// TwinCAT 3 PLC project TcUnitVerifier
// Title: TcUnit verifier
// Company: www.tcunit.org
// Author: Jakob Sagatowski and contributors
// ProjectVersion: 1.2.1.0
// Description: This project is can be used to verify the different functions of TcUnit. It has various test suites to test different functions in TcUnit. By making sure to comment out everything except the test suite that is interesting it is possible to test only the specific function of TcUnit that is interesting.
// ProgramVersion: 3.1.4022.7
// libraries:
//   SysDir, * (System)
//   SysFile, * (System)
//   Tc2_Standard, * (Beckhoff Automation GmbH)
//   Tc2_System, * (Beckhoff Automation GmbH)
//   Tc3_Module, * (Beckhoff Automation GmbH)
//   TcUnit, * (www.tcunit.org)
//   Base Interfaces,newest,System
// project tree:
//   / PlcTask.TcTTO
//   POUs/ FB_ProtectedVariables.TcPOU
//   Test/ FB_AdjustAssertFailureMessageToMaxAllowedLengthTest.TcPOU, FB_TestDurationMeasurement.TcPOU, FB_AnyPrimitiveTypes.TcPOU, FB_AnyToUnionValue.TcPOU, FB_ArrayPrimitiveTypes.TcPOU, FB_AssertCountExceedsMaxNumber.TcPOU, FB_AssertEveryFailedTestTwice.TcPOU, FB_AssertEveryFailedTestTwiceArrayVersion.TcPOU, FB_AssertTrueFalse.TcPOU, FB_CheckIfSpecificTestIsFinished.TcPOU, FB_CreateDisabledTest.TcPOU, FB_CreateFourTestsWithSameName.TcPOU, FB_EmptyAssertionMessage.TcPOU, FB_EmptyTestSuite.TcPOU, FB_ExtendedTestInformation.TcPOU, FB_MultipleAssertWithSameParametersInDifferentCyclesAndInSameTest.TcPOU, FB_MultipleAssertWithSameParametersInDifferentCyclesButWithDifferentTests.TcPOU, FB_MultipleAssertWithSameParametersInSameCycleWithSameTest.TcPOU, FB_SkipAssertionsWhenFinished.TcPOU, FB_PrimitiveTypes.TcPOU, FB_TestFileControl.TcPOU, FB_TestFinishedNamed.TcPOU, FB_TestNumberOfAssertionsCalculation.TcPOU, FB_TestStreamBuffer.TcPOU, FB_TestXmlControl.TcPOU, FB_WriteProtectedFunctions.TcPOU, FB_TestFinishedNamedDoesNotExist.TcPOU, PRG_TEST.TcPOU
//   Version/ Global_Version.TcGVL
// real-time tasks:
//   TASK PlcTask: cycle T#10ms, priority 20, ADS port 350

CONFIGURATION TcUnitVerifier
    RESOURCE PLC ON TwinCAT3
        TASK PlcTask(INTERVAL := T#10ms, PRIORITY := 20);
        PROGRAM PRG_TEST WITH PlcTask : PRG_TEST;
    END_RESOURCE
END_CONFIGURATION

// ---- Version/Global_Version.TcGVL
{attribute 'TcGenerated'}
{attribute 'no-analysis'}
{attribute 'linkalways'}
// This function has been automatically generated from the project information.
VAR_GLOBAL CONSTANT
	{attribute 'const_non_replaced'}
	stLibVersion_TcUnit_verifier : ST_LibVersion := (iMajor := 1, iMinor := 2, iBuild := 1, iRevision := 0, nFlags := 0, sVersion := '1.2.1.0');
END_VAR

// ---- Test/PRG_TEST.TcPOU
PROGRAM PRG_TEST
VAR
    PrimitiveTypes : FB_PrimitiveTypes;
    (* The FB_ExtendedTestInformation needs to be instantiated as the second test suite in order to get ID=1 as
       test suite identity, which is verified by the .NET-verifier *)
    ExtendedTestInformation : FB_ExtendedTestInformation;
    AssertTrueFalse : FB_AssertTrueFalse;
    AssertEveryFailedTestTwice : FB_AssertEveryFailedTestTwice;
    CreateFourTestsWithSameName : FB_CreateFourTestsWithSameName;
    ArrayPrimitiveTypes : FB_ArrayPrimitiveTypes;
    CreateDisabledTest : FB_CreateDisabledTest;
    AnyPrimitiveTypes : FB_AnyPrimitiveTypes;
    AssertEveryFailedTestTwiceArrayVersion : FB_AssertEveryFailedTestTwiceArrayVersion;
    AnyToUnionValue : FB_AnyToUnionValue;
    MultipleAssertWithSameParametersInSameCycleWithSameTest : FB_MultipleAssertWithSameParametersInSameCycleWithSameTest;
    MultipleAssertWithSameParametersInDifferentCyclesButWithDifferentTests : FB_MultipleAssertWithSameParametersInDifferentCyclesButWithDifferentTests;
    MultipleAssertWithSameParametersInDifferentCyclesAndInSameTest : FB_MultipleAssertWithSameParametersInDifferentCyclesAndInSameTest;
    SkipAssertionsWhenFinished : FB_SkipAssertionsWhenFinished;
    AdjustAssertFailureMessageToMaxAllowedLengthTest : FB_AdjustAssertFailureMessageToMaxAllowedLengthTest;
    EmptyTestSuite : FB_EmptyTestSuite;
    CheckIfSpecificTestIsFinished : FB_CheckIfSpecificTestIsFinished;
    WriteProtectedFunctions : FB_WriteProtectedFunctions;
    TestNumberOfAssertionsCalculation : FB_TestNumberOfAssertionsCalculation;
    TestDurationMeasurement : FB_TestDurationMeasurement;
    TestFileControl : FB_TestFileControl;
    TestXmlControl : FB_TestXmlControl;
    TestStreamBuffer : FB_TestStreamBuffer;
    TestFinishedNamed : FB_TestFinishedNamed;
    EmptyAssertionMessage : FB_EmptyAssertionMessage;
    AssertCountExceedsMaxNumber : FB_AssertCountExceedsMaxNumber;
    (* The testsuite below is not active, as it will make TcUnit to abort. Uncomment if you want
       to test the function of where a test with a name that doesn't exist is set to finished *)
    //TestFinishedNamedDoesNotExist : FB_TestFinishedNamedDoesNotExist;
END_VAR

(* There are two ways to run TcUnit test suites:
    1. The RUN() will run all the test suites in parallel
    2. The RUN_IN_SEQUENCE() will run the test suites in sequence (one-by-one, next one doesn't start until the previous one is finished)
    Only use one of them at a time
*)

TcUnit.RUN();
//TcUnit.RUN_IN_SEQUENCE(T#0MS);

END_PROGRAM

// ---- Test/FB_PrimitiveTypes.TcPOU
(*
    This testsuite tests the different assert-functions for all the different data types in TwinCAT.
    For every data type at least two different tests have been defined:
        1. One test that succeeds (Expected and actual are equal)
        2. One test that fails (Expected and actual are false).
*)
FUNCTION_BLOCK FB_PrimitiveTypes EXTENDS TcUnit.FB_TestSuite

Test_ANY_Equals();
Test_ANY_Differ_DataType();
Test_BOOL_Equals();
Test_BOOL_Differ();
Test_BYTE_Equals();
Test_BYTE_Differ();
Test_DATE_AND_TIME_Equals();
Test_DATE_AND_TIME_Differ();
Test_DATE_Equals();
Test_DATE_Differ();
Test_DINT_Equals();
Test_DINT_Differ();
Test_DWORD_Equals();
Test_DWORD_Differ();
Test_INT_Equals();
Test_INT_Differ();
Test_LINT_Equals();
Test_LINT_Differ();
Test_LREAL_Equals();
Test_LREAL_Differ();
Test_LTIME_Equals();
Test_LTIME_Differ();
Test_LWORD_Equals();
Test_LWORD_Differ();
Test_REAL_Equals();
Test_REAL_Differ();
Test_SINT_Equals();
Test_SINT_Differ();
Test_STRING_Equals();
Test_STRING_Differ();
Test_STRING_Differ2();
Test_STRING_Differ3();
Test_TIME_Equals();
Test_TIME_Differ();
Test_TIME_OF_DAY_Equals();
Test_TIME_OF_DAY_Differ();
Test_UDINT_Equals();
Test_UDINT_Differ();
Test_UINT_Equals();
Test_UINT_Differ();
Test_ULINT_Equals();
Test_ULINT_Differ();
Test_USINT_Equals();
Test_USINT_Differ();
Test_WORD_Equals();
Test_WORD_Differ();
Test_WSTRING_Equals();
Test_WSTRING_Differ();

METHOD PRIVATE Test_ANY_Differ_DataType
VAR
    a : INT := 5;
    b : UINT := 5;
END_VAR
TEST('Test_ANY_Differ_DataType');

AssertEquals(Expected := a,
             Actual := b,
             Message := 'Values differ');

TEST_FINISHED();
END_METHOD

METHOD PRIVATE Test_ANY_Equals
VAR
    a : INT := 5;
    b : INT := 5;
END_VAR
TEST('Test_ANY_Equals');

AssertEquals(Expected := a,
             Actual := b,
             Message := 'Values differ');

TEST_FINISHED();
END_METHOD

METHOD PRIVATE Test_BOOL_Differ
VAR
    a : BOOL := TRUE;
    b : BOOL := FALSE;
END_VAR
TEST('Test_BOOL_Differ');

TCUNIT_ADSLOGSTR(msgCtrlMask := ADSLOG_MSGTYPE_ERROR,
                 msgFmtStr := 'This is just a string %s',
                 strArg := '2');

AssertEquals_BOOL(Expected := a,
                  Actual := b,
                  Message := 'Values differ');

TEST_FINISHED();
END_METHOD

METHOD PRIVATE Test_BOOL_Equals
VAR
    a : BOOL := TRUE;
    b : BOOL := TRUE;
END_VAR
TEST('Test_BOOL_Equals');

TCUNIT_ADSLOGSTR(msgCtrlMask := ADSLOG_MSGTYPE_ERROR,
                 msgFmtStr := 'This is just a string %s',
                 strArg := '1');

AssertEquals_BOOL(Expected := a,
                  Actual := b,
                  Message := 'Values differ');

TEST_FINISHED();
END_METHOD

METHOD PRIVATE Test_BYTE_Differ
VAR
    a : BYTE := 16#AB;
    b : BYTE := 16#CD;
END_VAR
TEST('Test_BYTE_Differ');

AssertEquals_BYTE(Expected := a,
                  Actual := b,
                  Message := 'Values differ');

TEST_FINISHED();
END_METHOD

METHOD PRIVATE Test_BYTE_Equals
VAR
    a : BYTE := 16#CD;
    b : BYTE := 16#CD;
END_VAR
TEST('Test_BYTE_Equals');

AssertEquals_BYTE(Expected := a,
                  Actual := b,
                  Message := 'Values differ');
TEST_FINISHED();
END_METHOD

METHOD PRIVATE Test_DATE_AND_TIME_Differ
VAR
    a : DATE_AND_TIME := DATE_AND_TIME#1996-05-06-15:36:30;
    b : DATE_AND_TIME := DATE_AND_TIME#1972-03-29-00:00:00;
END_VAR
TEST('Test_DATE_AND_TIME_Differ');

AssertEquals_DATE_AND_TIME(Expected := a,
                           Actual := b,
                           Message := 'Values differ');

TEST_FINISHED();
END_METHOD

METHOD PRIVATE Test_DATE_AND_TIME_Equals
VAR
    a : DATE_AND_TIME := DATE_AND_TIME#2019-01-20-13:54:30;
    b : DATE_AND_TIME := DATE_AND_TIME#2019-01-20-13:54:30;
END_VAR
TEST('Test_DATE_AND_TIME_Equals');

AssertEquals_DATE_AND_TIME(Expected := a,
                           Actual := b,
                           Message := 'Values differ');

TEST_FINISHED();
END_METHOD

METHOD PRIVATE Test_DATE_Differ
VAR
    a : DATE := DATE#1996-05-06;
    b : DATE := DATE#2019-01-20;
END_VAR
TEST('Test_DATE_Differ');

AssertEquals_DATE(Expected := a,
                  Actual := b,
                  Message := 'Values differ');

TEST_FINISHED();
END_METHOD

METHOD PRIVATE Test_DATE_Equals
VAR
    a : DATE := DATE#1996-05-06;
    b : DATE := DATE#1996-05-06;
END_VAR
TEST('Test_DATE_Equals');

AssertEquals_DATE(Expected := a,
                  Actual := b,
                  Message := 'Values differ');

TEST_FINISHED();
END_METHOD

METHOD PRIVATE Test_DINT_Differ
VAR
    a : DINT := -55555;
    b : DINT := 70000;
END_VAR
TEST('Test_DINT_Differ');

AssertEquals_DINT(Expected := a,
                  Actual := b,
                  Message := 'Values differ');

TEST_FINISHED();
END_METHOD

METHOD PRIVATE Test_DINT_Equals
VAR
    a : DINT := -80000;
    b : DINT := -80000;
END_VAR
TEST('Test_DINT_Equals');

AssertEquals_DINT(Expected := a,
                  Actual := b,
                  Message := 'Values differ');

TEST_FINISHED();
END_METHOD

METHOD PRIVATE Test_DWORD_Differ
VAR
    a : DWORD := 16#12345678;
    b : DWORD := 16#90ABCDEF;
END_VAR
TEST('Test_DWORD_Differ');

TCUNIT_ADSLOGSTR(msgCtrlMask := ADSLOG_MSGTYPE_HINT,
                 msgFmtStr := 'This is just a string %s',
                 strArg := '4');

AssertEquals_DWORD(Expected := a,
                   Actual := b,
                   Message := 'Values differ');

TEST_FINISHED();
END_METHOD

METHOD PRIVATE Test_DWORD_Equals
VAR
    a : DWORD := 16#7890ABCD;
    b : DWORD := 16#7890ABCD;
END_VAR
TEST('Test_DWORD_Equals');

TCUNIT_ADSLOGSTR(msgCtrlMask := ADSLOG_MSGTYPE_HINT,
                 msgFmtStr := 'This is just a string %s',
                 strArg := '3');

AssertEquals_DWORD(Expected := a,
                   Actual := b,
                   Message := 'Values differ');

TEST_FINISHED();
END_METHOD

METHOD PRIVATE Test_INT_Differ
VAR
    a : INT := -32000;
    b : INT := 15423;
END_VAR
TEST('Test_INT_Differ');

AssertEquals_INT(Expected := a,
                 Actual := b,
                 Message := 'Values differ');

TEST_FINISHED();
END_METHOD

METHOD PRIVATE Test_INT_Equals
VAR
    a : INT := -12345;
    b : INT := -12345;
END_VAR
TEST('Test_INT_Equals');

AssertEquals_INT(Expected := a,
                 Actual := b,
                 Message := 'Values differ');

TEST_FINISHED();
END_METHOD

METHOD PRIVATE Test_LINT_Differ
VAR
    a : LINT := -451416345;
    b : LINT := 589532453;
END_VAR
TEST('Test_LINT_Differ');

AssertEquals_LINT(Expected := a,
                  Actual := b,
                  Message := 'Values differ');

TEST_FINISHED();
END_METHOD

METHOD PRIVATE Test_LINT_Equals
VAR
    a : LINT := -123456789;
    b : LINT := -123456789;
END_VAR
TEST('Test_LINT_Equals');

AssertEquals_LINT(Expected := a,
                  Actual := b,
                  Message := 'Values differ');

TEST_FINISHED();
END_METHOD

METHOD PRIVATE Test_LREAL_Differ
VAR
    a : LREAL := 1234567.89;
    b : LREAL := 1234567.76;
    c : LREAL := 0.0;
END_VAR
TEST('Test_LREAL_Differ');

AssertEquals_LREAL(Expected := a,
                   Actual := b,
                   Delta := 0.1,
                   Message := 'Values a and b differ');

MEMSET (ADR(c), 255, SIZEOF(c));

AssertEquals_LREAL(Expected := a,
                   Actual := c,
                   Delta := 0.1,
                   Message := 'Values a and c differ');

TEST_FINISHED();
END_METHOD

METHOD PRIVATE Test_LREAL_Equals
VAR
    a : LREAL := 1234567.89;
    b : LREAL := 1234567.76;
END_VAR
TEST('Test_LREAL_Equals');

AssertEquals_LREAL(Expected := a,
                   Actual := b,
                   Delta := 0.2,
                   Message := 'Values differ');

TEST_FINISHED();
END_METHOD

METHOD PRIVATE Test_LTIME_Differ
VAR
    a : LTIME := LTIME#213503D23H34M33S709MS551US615NS;
    b : LTIME := LTIME#1000D15H23M12S34MS2US44NS;
END_VAR
TEST('Test_LTIME_Differ');

AssertEquals_LTIME(Expected := a,
                   Actual := b,
                   Message := 'Values differ');

TEST_FINISHED();
END_METHOD

METHOD PRIVATE Test_LTIME_Equals
VAR
    a : LTIME := LTIME#213503D23H34M33S709MS551US615NS;
    b : LTIME := LTIME#213503D23H34M33S709MS551US615NS;
END_VAR
TEST('Test_LTIME_Equals');

AssertEquals_LTIME(Expected := a,
                   Actual := b,
                   Message := 'Values differ');

TEST_FINISHED();
END_METHOD

METHOD PRIVATE Test_LWORD_Differ
VAR
    a : LWORD := 16#0123656789ABCBEC;
    b : LWORD := 16#0123256789ABCAEE;
END_VAR
TEST('Test_LWORD_Differ');

AssertEquals_LWORD(Expected := a,
                   Actual := b,
                   Message := 'Values differ');

TEST_FINISHED();
END_METHOD

METHOD PRIVATE Test_LWORD_Equals
VAR
    a : LWORD := 16#0123456789ABCDEF;
    b : LWORD := 16#0123456789ABCDEF;
END_VAR
TEST('Test_LWORD_Equals');

AssertEquals_LWORD(Expected := a,
                   Actual := b,
                   Message := 'Values differ');

TEST_FINISHED();
END_METHOD

METHOD PRIVATE Test_REAL_Differ
VAR
    a : REAL := 1234.5;
    b : REAL := 1234.4;
    c : REAL := 0.0;
END_VAR
TEST('Test_REAL_Differ');

TCUNIT_ADSLOGSTR(msgCtrlMask := ADSLOG_MSGTYPE_WARN,
                 msgFmtStr := 'This is just a string %s',
                 strArg := '6');

AssertEquals_REAL(Expected := a,
                  Actual := b,
                  Delta := 0.05,
                  Message := 'Values a and b differ');

MEMSET (ADR(c), 255, SIZEOF(c));

AssertEquals_REAL(Expected := a,
                  Actual := c,
                  Delta := 0.1,
                  Message := 'Values a and c differ');

TEST_FINISHED();
END_METHOD

METHOD PRIVATE Test_REAL_Equals
VAR
    a : REAL := 1234.5;
    b : REAL := 1234.4;
END_VAR
TEST('Test_REAL_Equals');

TCUNIT_ADSLOGSTR(msgCtrlMask := ADSLOG_MSGTYPE_WARN,
                 msgFmtStr := 'This is just a string %s',
                 strArg := '5');

AssertEquals_REAL(Expected := a,
                  Actual := b,
                  Delta := 0.1,
                  Message := 'Values differ');

TEST_FINISHED();
END_METHOD

METHOD PRIVATE Test_SINT_Differ
VAR
    a : SINT := 127;
    b : SINT := -30;
END_VAR
TEST('Test_SINT_Differ');

AssertEquals_SINT(Expected := a,
                  Actual := b,
                  Message := 'Values differ');

TEST_FINISHED();
END_METHOD

METHOD PRIVATE Test_SINT_Equals
VAR
    a : SINT := -128;
    b : SINT := -128;
END_VAR
TEST('Test_SINT_Equals');

AssertEquals_SINT(Expected := a,
                  Actual := b,
                  Message := 'Values differ');

TEST_FINISHED();
END_METHOD

METHOD PRIVATE Test_STRING_Differ
VAR
    a : STRING := 'This is a string';
    b : STRING := 'This is another string';
END_VAR
TEST('Test_STRING_Differ');

AssertEquals_STRING(Expected := a,
                    Actual := b,
                    Message := 'Values differ');

TEST_FINISHED();
END_METHOD

METHOD PRIVATE Test_STRING_Differ2
VAR
    a : STRING := '';
    b : STRING := 'This string is not empty';
END_VAR
TEST('Test_STRING_Differ2');

AssertEquals_STRING(Expected := a,
                    Actual := b,
                    Message := 'Values differ');

TEST_FINISHED();
END_METHOD

METHOD PRIVATE Test_STRING_Differ3
VAR
    a : STRING := 'This string is not empty';
    b : STRING := '';
END_VAR
TEST('Test_STRING_Differ3');

AssertEquals_STRING(Expected := a,
                    Actual := b,
                    Message := 'Values differ');

TEST_FINISHED();
END_METHOD

METHOD PRIVATE Test_STRING_Equals
VAR
    a : STRING := 'Hello there';
    b : STRING := 'Hello there';
END_VAR
TEST('Test_STRING_Equals');

AssertEquals_STRING(Expected := a,
                    Actual := b,
                    Message := 'Values differ');

TEST_FINISHED();
END_METHOD

METHOD PRIVATE Test_TIME_Differ
VAR
    a : TIME := T#12H34M15S10MS;
    b : TIME := T#11H34M13S244MS;
END_VAR
TEST('Test_TIME_Differ');

AssertEquals_TIME(Expected := a,
                  Actual := b,
                  Message := 'Values differ');

TEST_FINISHED();
END_METHOD

METHOD PRIVATE Test_TIME_Equals
VAR
    a : TIME := T#11H34M13S244MS;
    b : TIME := T#11H34M13S244MS;
END_VAR
TEST('Test_TIME_Equals');

AssertEquals_TIME(Expected := a,
                  Actual := b,
                  Message := 'Values differ');

TEST_FINISHED();
END_METHOD

METHOD PRIVATE Test_TIME_OF_DAY_Differ
VAR
    a : TIME_OF_DAY := TIME_OF_DAY#15:36:30.123;
    b : TIME_OF_DAY := TIME_OF_DAY#06:21:11.492;
END_VAR
TEST('Test_TIME_OF_DAY_Differ');

AssertEquals_TIME_OF_DAY(Expected := a,
                         Actual := b,
                         Message := 'Values differ');

TEST_FINISHED();
END_METHOD

METHOD PRIVATE Test_TIME_OF_DAY_Equals
VAR
    a : TIME_OF_DAY := TIME_OF_DAY#06:21:11.492;
    b : TIME_OF_DAY := TIME_OF_DAY#06:21:11.492;
END_VAR
TEST('Test_TIME_OF_DAY_Equals');

AssertEquals_TIME_OF_DAY(Expected := a,
                         Actual := b,
                         Message := 'Values differ');

TEST_FINISHED();
END_METHOD

METHOD PRIVATE Test_UDINT_Differ
VAR
    a : UDINT := 34124214;
    b : UDINT := 52343244;
END_VAR
TEST('Test_UDINT_Differ');

AssertEquals_UDINT(Expected := a,
                   Actual := b,
                   Message := 'Values differ');

TEST_FINISHED();
END_METHOD

METHOD PRIVATE Test_UDINT_Equals
VAR
    a : UDINT := 21845123;
    b : UDINT := 21845123;
END_VAR
TEST('Test_UDINT_Equals');

AssertEquals_UDINT(Expected := a,
                   Actual := b,
                   Message := 'Values differ');

TEST_FINISHED();
END_METHOD

METHOD PRIVATE Test_UINT_Differ
VAR
    a : UINT := 64322;
    b : UINT := 32312;
END_VAR
TEST('Test_UINT_Differ');

AssertEquals_UINT(Expected := a,
                  Actual := b,
                  Message := 'Values differ');

TEST_FINISHED();
END_METHOD

METHOD PRIVATE Test_UINT_Equals
VAR
    a : UINT := 65535;
    b : UINT := 65535;
END_VAR
TEST('Test_UINT_Equals');

AssertEquals_UINT(Expected := a,
                  Actual := b,
                  Message := 'Values differ');

TEST_FINISHED();
END_METHOD

METHOD PRIVATE Test_ULINT_Differ
VAR
    a : ULINT := 10000;
    b : ULINT := 53685437234;
END_VAR
TEST('Test_ULINT_Differ');

AssertEquals_ULINT(Expected := a,
                   Actual := b,
                   Message := 'Values differ');

TEST_FINISHED();
END_METHOD

METHOD PRIVATE Test_ULINT_Equals
VAR
    a : ULINT := 45683838383;
    b : ULINT := 45683838383;
END_VAR
TEST('Test_ULINT_Equals');

AssertEquals_ULINT(Expected := a,
                   Actual := b,
                   Message := 'Values differ');

TEST_FINISHED();
END_METHOD

METHOD PRIVATE Test_USINT_Differ
VAR
    a : USINT := 3;
    b : USINT := 7;
END_VAR
TEST('Test_USINT_Differ');

AssertEquals_USINT(Expected := a,
                   Actual := b,
                   Message := 'Values differ');

TEST_FINISHED();
END_METHOD

METHOD PRIVATE Test_USINT_Equals
VAR
    a : USINT := 5;
    b : USINT := 5;
END_VAR
TEST('Test_USINT_Equals');

AssertEquals_USINT(Expected := a,
                   Actual := b,
                   Message := 'Values differ');

TEST_FINISHED();
END_METHOD

METHOD PRIVATE Test_WORD_Differ
VAR
    a : WORD := 16#EF01;
    b : WORD := 16#2345;
END_VAR
TEST('Test_WORD_Differ');

AssertEquals_WORD(Expected := a,
                  Actual := b,
                  Message := 'Values differ');

TEST_FINISHED();
END_METHOD

METHOD PRIVATE Test_WORD_Equals
VAR
    a : WORD := 16#ABCD;
    b : WORD := 16#ABCD;
END_VAR
TEST('Test_WORD_Equals');

AssertEquals_WORD(Expected := a,
                  Actual := b,
                  Message := 'Values differ');

TEST_FINISHED();
END_METHOD

METHOD PRIVATE Test_WSTRING_Differ
VAR
    a : WSTRING := "äö";
    b : WSTRING := "æåŅ";
END_VAR
TEST('Test_WSTRING_Differ');

AssertEquals_WSTRING(Expected := a,
                     Actual := b,
                     Message := 'Values differ');

TEST_FINISHED();
END_METHOD

METHOD PRIVATE Test_WSTRING_Equals
VAR
    a : WSTRING := "ŏŜŢ";
    b : WSTRING := "ŏŜŢ";
END_VAR
TEST('Test_WSTRING_Equals');

AssertEquals_WSTRING(Expected := a,
                     Actual := b,
                     Message := 'Values differ');

TEST_FINISHED();
END_METHOD

END_FUNCTION_BLOCK

// ---- Test/FB_ExtendedTestInformation.TcPOU
(* This test suite makes sure to create different variants of tests that will produce various extended logs, i.e. the
   ADS-logs that provide information on how many tests have finished/are successful within the test suites.
   This test suite needs to be instantiated as the second test suite in the order in order to get the ID=1 as identity. *)
FUNCTION_BLOCK FB_ExtendedTestInformation EXTENDS TcUnit.FB_TestSuite

Test_ExtendedTestInformation_BOOL_AssertFailed();
Test_ExtendedTestInformation_BOOL_AssertSuccess();
Test_ExtendedTestInformation_BYTE_TwoFailedAsserts();
Test_ExtendedTestInformation_LINT_AssertFailed();
Test_ExtendedTestInformation_LINT_AssertSuccess();

METHOD PRIVATE Test_ExtendedTestInformation_BOOL_AssertFailed
VAR
    a : BOOL := TRUE;
    b : BOOL := FALSE;
END_VAR
TEST('Test_ExtendedTestInformation_BOOL_AssertFailed');

AssertEquals_BOOL(Expected := a,
                  Actual := b,
                  Message := 'Extendedinformation values differ BOOL failure');

TEST_FINISHED();
END_METHOD

METHOD PRIVATE Test_ExtendedTestInformation_BOOL_AssertSuccess
VAR
    a : BOOL := TRUE;
    b : BOOL := TRUE;
END_VAR
TEST('Test_ExtendedTestInformation_BOOL_AssertSuccess');

AssertEquals_BOOL(Expected := a,
                  Actual := b,
                  Message := 'Extendedinformation values differ BOOL success');

TEST_FINISHED();
END_METHOD

METHOD PRIVATE Test_ExtendedTestInformation_BYTE_TwoFailedAsserts
VAR
    a : BYTE := 16#AB;
    b : BYTE := 16#CD;
    c : BYTE := 16#EF;
    d : BYTE := 16#01;
END_VAR
TEST('Test_ExtendedTestInformation_BYTE_TwoFailedAsserts');

AssertEquals_BYTE(Expected := a,
                  Actual := b,
                  Message := 'Extendedinformation values differ BYTE1');

AssertEquals_BYTE(Expected := c,
                  Actual := d,
                  Message := 'Extendedinformation values differ BYTE2');

TEST_FINISHED();
END_METHOD

METHOD PRIVATE Test_ExtendedTestInformation_LINT_AssertFailed
VAR
    a : LINT := -451416345;
    b : LINT := 589532453;
END_VAR
TEST('Test_ExtendedTestInformation_LINT_AssertFailed');

AssertEquals_LINT(Expected := a,
                  Actual := b,
                  Message := 'Extendedinformation values differ LINT failure');

TEST_FINISHED();
END_METHOD

METHOD PRIVATE Test_ExtendedTestInformation_LINT_AssertSuccess
VAR
    a : LINT := -123456789;
    b : LINT := -123456789;
END_VAR
TEST('Test_ExtendedTestInformation_LINT_AssertSuccess');

AssertEquals_LINT(Expected := a,
                  Actual := b,
                  Message := 'Extendedinformation values differ LINT success');

TEST_FINISHED();
END_METHOD

END_FUNCTION_BLOCK

// ---- Test/FB_AssertTrueFalse.TcPOU
(* 
    This testsuite verifies that the Assert_True and Assert_False methods do what they are supposed to. It does so
    by making sure that every assert-method (assert_true & assert_false) does both one failing and one successful
    assert.
*)
FUNCTION_BLOCK FB_AssertTrueFalse EXTENDS TcUnit.FB_TestSuite

AssertThatINTsAreEqual();
AssertThatINTsAreNotEqual();
AssertThatWORDsAreEqual();
AssertThatWORDsAreNotEqual();

METHOD PRIVATE AssertThatINTsAreEqual
VAR
    a : INT := -33;
    b : INT := -44;
END_VAR
TEST('AssertThatINTsAreEqual');

AssertFalse(Condition := (a <> b),
            Message := 'INTs are equal');

TEST_FINISHED();
END_METHOD

METHOD PRIVATE AssertThatINTsAreNotEqual
VAR
    a : INT := -33;
    b : INT := -44;
END_VAR
TEST('AssertThatINTsAreNotEqual');

AssertFalse(Condition := (a = b),
            Message := 'INTs are equal');

TEST_FINISHED();
END_METHOD

METHOD PRIVATE AssertThatWORDsAreEqual
VAR
    a : WORD := 16#ABCD;
    b : WORD := 16#0123;
END_VAR
TEST('AssertThatWORDsAreEqual');

AssertTrue(Condition := (a = b),
           Message := 'WORDs are not equal');

TEST_FINISHED();
END_METHOD

METHOD PRIVATE AssertThatWORDsAreNotEqual
VAR
    a : WORD := 16#ABCD;
    b : WORD := 16#0123;
END_VAR
TEST('AssertThatWORDsAreNotEqual');

AssertTrue(Condition := (a <> b),
           Message := 'WORDs are equal');

TEST_FINISHED();
END_METHOD

END_FUNCTION_BLOCK

// ---- Test/FB_AssertEveryFailedTestTwice.TcPOU
(*
    In this testsuite we are running the same testcase over two cycles, and thus calling every assert method twice.
    This is in order to verify that we don't print every FAILED assert twice.
*)
FUNCTION_BLOCK FB_AssertEveryFailedTestTwice EXTENDS TcUnit.FB_TestSuite
VAR
    AssertCount : USINT := 0;
END_VAR

TwiceAssertCall();

METHOD PRIVATE TwiceAssertCall
VAR
    aANY : INT := 55;
    bANY : INT := 77;

    aBOOL : BOOL := TRUE;
    bBOOL : BOOL := FALSE;

    aBYTE : BYTE := 16#AB;
    bBYTE : BYTE := 16#BA;

    aDATE : DATE := DATE#1996-05-06;
    bDATE : DATE := DATE#2019-01-20;

    aDATE_AND_TIME : DATE_AND_TIME := DATE_AND_TIME#1996-05-06-15:36:30;
    bDATE_AND_TIME : DATE_AND_TIME := DATE_AND_TIME#1972-03-29-00:00:00;

    aDINT : DINT := 4444;
    bDINT : DINT := 3333;

    aDWORD : DWORD := 16#AAAAAAAA;
    bDWORD : DWORD := 16#BBBBBBBB;

    aINT : INT := 30000;
    bINT : INT := 32000;

    aLINT : LINT := 50000;
    bLINT : LINT := 50001;

    aLREAL : LREAL := 33.3;
    bLREAL : LREAL := 44.4;

    aLTIME : LTIME := LTIME#213503D23H34M33S709MS551US615NS;
    bLTIME : LTIME := LTIME#1000D15H23M12S34MS2US44NS;

    aLWORD : LWORD := 16#AAAAAAAAAAAAAAAA;
    bLWORD : LWORD := 16#BBBBBBBBBBBBBBBB;

    aREAL : REAL := 44.4;
    bREAL : REAL := 22.2;

    aSINT : SINT := 99;
    bSINT : SINT := 10;

    aSTRING : STRING := 'Hello world';
    bSTRING : STRING := 'Hey there';

    aUDINT : UDINT := 249494994;
    bUDINT : UDINT := 1223;

    aUINT : UINT := 3444;
    bUINT : UINT := 3445;

    aULINT : ULINT := 789234475;
    bULINT : ULINT := 34523327234;

    aUSINT : USINT := 34;
    bUSINT : USINT := 36;

    aTIME : TIME := T#12H34M15S10MS;
    bTIME : TIME := T#11H34M13S244MS;

    aTIME_OF_DAY : TIME_OF_DAY := TIME_OF_DAY#15:36:30.123;
    bTIME_OF_DAY : TIME_OF_DAY := TIME_OF_DAY#06:21:11.492;

    aWORD : WORD := 16#ABCD;
    bWORD : WORD := 16#89EF;

	aWSTRING : WSTRING := "åäöĦ";
    bWSTRING : WSTRING := "åäöŅ";
END_VAR
TEST('TwiceAssertCall');

AssertEquals(Expected := aANY,
             Actual := bANY,
             Message := 'Not equal ANY');

AssertEquals_BOOL(Expected := aBOOL,
                  Actual := bBOOL,
                  Message := 'Not equal BOOL');

AssertEquals_BYTE(Expected := aBYTE,
                  Actual := bBYTE,
                  Message := 'Not equal BYTE');

AssertEquals_DATE(Expected := aDATE,
                  Actual := bDATE,
                  Message := 'Not equal DATE');

AssertEquals_DATE_AND_TIME(Expected := aDATE_AND_TIME,
                           Actual := bDATE_AND_TIME,
                           Message := 'Not equal DATE_AND_TIME');

AssertEquals_DINT(Expected := aDINT,
                  Actual := bDINT,
                  Message := 'Not equal DINT');

AssertEquals_DWORD(Expected := aDWORD,
                   Actual := bDWORD,
                   Message := 'Not equal DWORD');

AssertEquals_INT(Expected := aINT,
                 Actual := bINT,
                 Message := 'Not equal INT');

AssertEquals_LINT(Expected := aLINT,
                  Actual := bLINT,
                  Message := 'Not equal LINT');

AssertEquals_LREAL(Expected := aLREAL,
                   Actual := bLREAL,
                   Delta := 0.1,
                   Message := 'Not equal LREAL');

AssertEquals_LTIME(Expected := aLTIME,
                   Actual := bLTIME,
                   Message := 'Not equal LTIME');

AssertEquals_LWORD(Expected := aLWORD,
                   Actual := bLWORD,
                   Message := 'Not equal LWORD');

AssertEquals_REAL(Expected := aREAL,
                  Actual := bREAL,
                  Delta := 0.1,
                  Message := 'Not equal REAL');

AssertEquals_SINT(Expected := aSINT,
                  Actual := bSINT,
                  Message := 'Not equal SINT');

AssertEquals_STRING(Expected := aSTRING,
                    Actual := bSTRING,
                    Message := 'Not equal STRING');

AssertEquals_UDINT(Expected := aUDINT,
                   Actual := bUDINT,
                   Message := 'Not equal UDINT');

AssertEquals_UINT(Expected := aUINT,
                  Actual := bUINT,
                  Message := 'Not equal UINT');

AssertEquals_ULINT(Expected := aULINT,
                   Actual := bULINT,
                   Message := 'Not equal ULINT');

AssertEquals_USINT(Expected := aUSINT,
                   Actual := bUSINT,
                   Message := 'Not equal USINT');

AssertEquals_TIME(Expected := aTIME,
                  Actual := bTIME,
                  Message := 'Not equal TIME');

AssertEquals_TIME_OF_DAY(Expected := aTIME_OF_DAY,
                         Actual := bTIME_OF_DAY,
                         Message := 'Not equal TIME_OF_DAY');

AssertEquals_WORD(Expected := aWORD,
                  Actual := bWORD,
                  Message := 'Not equal WORD');

AssertEquals_WSTRING(Expected := aWSTRING,
                     Actual := bWSTRING,
                     Message := 'Not equal WSTRING');

AssertCount := AssertCount + 1;
IF AssertCount = 2 THEN
    TEST_FINISHED();
END_IF
END_METHOD

END_FUNCTION_BLOCK

// ---- Test/FB_CreateFourTestsWithSameName.TcPOU
(*
    This testsuite creates four tests in the same testsuite with the same name. Every test in a testsuite should have
    an unique name. Every assert should be ignored if a duplicate test is being run.
*)
FUNCTION_BLOCK FB_CreateFourTestsWithSameName EXTENDS TcUnit.FB_TestSuite

TestOne();
TestOne_Again();
TestOne_AgainAgain();
TestOne_AgainAgainAgain();

METHOD PRIVATE TestOne
VAR
    a : INT := 55;
    b : INT := 55;
END_VAR
TEST('TestOne');

AssertEquals_INT(Expected := a,
                 Actual := b,
                 Message := 'A does not equal B');

TEST_FINISHED();
END_METHOD

METHOD PRIVATE TestOne_Again
VAR
    a : INT := 55;
    b : INT := 54;
END_VAR
TEST('TestOne');

AssertEquals_INT(Expected := a,
                 Actual := b,
                 Message := 'A does not equal B again');

TEST_FINISHED();
END_METHOD

METHOD PRIVATE TestOne_AgainAgain
VAR
    a : INT := 55;
    b : INT := 55;
END_VAR
TEST('TestOne');

AssertEquals_INT(Expected := a,
                 Actual := b,
                 Message := 'A does not equal B again');

TEST_FINISHED();
END_METHOD

METHOD PRIVATE TestOne_AgainAgainAgain
VAR
    a : INT := 55;
    b : INT := 55;
END_VAR
TEST('TestOne');

AssertEquals_INT(Expected := a,
                 Actual := b,
                 Message := 'A does not equal B again');

TEST_FINISHED();
END_METHOD

END_FUNCTION_BLOCK

// ---- Test/FB_ArrayPrimitiveTypes.TcPOU
(*
    This testsuite tests the different assert-functions for all the different type of arrays (varying by the different
    data types that are available in TwinCAT). For every type of array (BOOL, BYTE, INT etc.) at least three different
    tests have been defined:
        1. One test that succeeds, where the data and size of the arrays are matching
        2. One test that fails, where the size of the arrays differs
        3. One test that fails, where the content of the array differs
*)
FUNCTION_BLOCK FB_ArrayPrimitiveTypes EXTENDS TcUnit.FB_TestSuite

Test_BOOL_Array_Equals();
Test_BOOL_Array_DifferInSize();
Test_BOOL_Array_DifferInContent();
Test_BYTE_Array_Equals();
Test_BYTE_Array_DifferInSize();
Test_BYTE_Array_DifferInContent();
Test_DINT_Array_Equals();
Test_DINT_Array_DifferInSize();
Test_DINT_Array_DifferInContent();
Test_DWORD_Array_Equals();
Test_DWORD_Array_DifferInSize();
Test_DWORD_Array_DifferInContent();
Test_INT_Array_Equals();
Test_INT_Array_DifferInSize();
Test_INT_Array_DifferInContent();
Test_LINT_Array_Equals();
Test_LINT_Array_DifferInSize();
Test_LINT_Array_DifferInContent();
Test_LREAL_Array_Equals();
Test_LREAL_Array_DifferInSize();
Test_LREAL_Array_DifferInContent();
Test_LREAL_Array2d_Equals();
Test_LREAL_Array2d_DifferInSize_D1();
Test_LREAL_Array2d_DifferInSize_D2();
Test_LREAL_Array2d_DifferInContent_LBOUND();
Test_LREAL_Array2d_DifferInContent_Middle();
Test_LREAL_Array2d_DifferInContent_UBOUND();
Test_LREAL_Array3d_Equals();
Test_LREAL_Array3d_DifferInSize_D1();
Test_LREAL_Array3d_DifferInSize_D2();
Test_LREAL_Array3d_DifferInSize_D3();
Test_LREAL_Array3d_DifferInContent_LBOUND();
Test_LREAL_Array3d_DifferInContent_Middle();
Test_LREAL_Array3d_DifferInContent_UBOUND();
Test_LWORD_Array_Equals();
Test_LWORD_Array_DifferInSize();
Test_LWORD_Array_DifferInContent();
Test_REAL_Array_Equals();
Test_REAL_Array_DifferInSize();
Test_REAL_Array_DifferInContent();
Test_REAL_Array2d_Equals();
Test_REAL_Array2d_DifferInSize_D1();
Test_REAL_Array2d_DifferInSize_D2();
Test_REAL_Array2d_DifferInContent_LBOUND();
Test_REAL_Array2d_DifferInContent_Middle();
Test_REAL_Array2d_DifferInContent_UBOUND();
Test_REAL_Array3d_Equals();
Test_REAL_Array3d_DifferInSize_D1();
Test_REAL_Array3d_DifferInSize_D2();
Test_REAL_Array3d_DifferInSize_D3();
Test_REAL_Array3d_DifferInContent_LBOUND();
Test_REAL_Array3d_DifferInContent_Middle();
Test_REAL_Array3d_DifferInContent_UBOUND();
Test_SINT_Array_Equals();
Test_SINT_Array_DifferInSize();
Test_SINT_Array_DifferInContent();
Test_UDINT_Array_Equals();
Test_UDINT_Array_DifferInSize();
Test_UDINT_Array_DifferInContent();
Test_UINT_Array_Equals();
Test_UINT_Array_DifferInSize();
Test_UINT_Array_DifferInContent();
Test_ULINT_Array_Equals();
Test_ULINT_Array_DifferInSize();
Test_ULINT_Array_DifferInContent();
Test_USINT_Array_Equals();
Test_USINT_Array_DifferInSize();
Test_USINT_Array_DifferInContent();
Test_WORD_Array_Equals();
Test_WORD_Array_DifferInSize();
Test_WORD_Array_DifferInContent();

METHOD PRIVATE Test_BOOL_Array_DifferInContent
VAR
    a : ARRAY[0..5] OF BOOL := [TRUE, TRUE, FALSE, TRUE, FALSE, TRUE];
    b : ARRAY[0..5] OF BOOL := [TRUE, TRUE, TRUE, TRUE, FALSE, FALSE];
END_VAR
TEST('Test_BOOL_Array_DifferInContent');

AssertArrayEquals_BOOL(Expecteds := a,
                       Actuals := b,
                       Message := 'Arrays differ');

TEST_FINISHED();
END_METHOD

METHOD PRIVATE Test_BOOL_Array_DifferInSize
VAR
    a : ARRAY[1..6] OF BOOL := [TRUE, TRUE, TRUE, TRUE, TRUE, TRUE];
    b : ARRAY[1..4] OF BOOL := [TRUE, TRUE, TRUE, TRUE];
END_VAR
TEST('Test_BOOL_Array_DifferInSize');

TCUNIT_ADSLOGSTR(msgCtrlMask := ADSLOG_MSGTYPE_HINT,
                 msgFmtStr := 'This is just a string %s',
                 strArg := '8');

AssertArrayEquals_BOOL(Expecteds := a,
                       Actuals := b,
                       Message := 'Arrays differ');

TEST_FINISHED();
END_METHOD

METHOD PRIVATE Test_BOOL_Array_Equals
VAR
    a : ARRAY[1..5] OF BOOL := [TRUE, FALSE, TRUE, FALSE, TRUE];
    b : ARRAY[1..5] OF BOOL := [TRUE, FALSE, TRUE, FALSE, TRUE];
END_VAR
TEST('Test_BOOL_Array_Equals');

TCUNIT_ADSLOGSTR(msgCtrlMask := ADSLOG_MSGTYPE_HINT,
                 msgFmtStr := 'This is just a string %s',
                 strArg := '7');

AssertArrayEquals_BOOL(Expecteds := a,
                       Actuals := b,
                       Message := 'Arrays differ');

TEST_FINISHED();
END_METHOD

METHOD PRIVATE Test_BYTE_Array_DifferInContent
VAR
    a : ARRAY[0..3] OF BYTE := [16#AB, 16#AA, 16#BB, 16#89];
    b : ARRAY[0..3] OF BYTE := [16#AB, 16#CD, 16#BB, 16#89];
END_VAR
TEST('Test_BYTE_Array_DifferInContent');

AssertArrayEquals_BYTE(Expecteds := a,
                       Actuals := b,
                       Message := 'Arrays differ');

TEST_FINISHED();
END_METHOD

METHOD PRIVATE Test_BYTE_Array_DifferInSize
VAR
    a : ARRAY[1..2] OF BYTE := [16#AB, 16#CD];
    b : ARRAY[1..5] OF BYTE := [16#AB, 16#CD, 16#EF, 16#01, 16#23];
END_VAR
TEST('Test_BYTE_Array_DifferInSize');

AssertArrayEquals_BYTE(Expecteds := a,
                       Actuals := b,
                       Message := 'Arrays differ');

TEST_FINISHED();
END_METHOD

METHOD PRIVATE Test_BYTE_Array_Equals
VAR
    a : ARRAY[1..3] OF BYTE := [16#FD, 16#34, 16#9E];
    b : ARRAY[1..3] OF BYTE := [16#FD, 16#34, 16#9E];
END_VAR
TEST('Test_BYTE_Array_Equals');

AssertArrayEquals_BYTE(Expecteds := a,
                       Actuals := b,
                       Message := 'Arrays differ');

TEST_FINISHED();
END_METHOD

METHOD PRIVATE Test_DINT_Array_DifferInContent
VAR
    a : ARRAY[3..5] OF DINT := [-4746, -2147483645, 0];
    b : ARRAY[3..5] OF DINT := [-4746, -2147483641, 0];
END_VAR
TEST('Test_DINT_Array_DifferInContent');

AssertArrayEquals_DINT(Expecteds := a,
                       Actuals := b,
                       Message := 'Arrays differ');

TEST_FINISHED();
END_METHOD

METHOD PRIVATE Test_DINT_Array_DifferInSize
VAR
    a : ARRAY[3..4] OF DINT := [-11, 2147483647];
    b : ARRAY[4..6] OF DINT := [-11, 2147483647, 0];
END_VAR
TEST('Test_DINT_Array_DifferInSize');

AssertArrayEquals_DINT(Expecteds := a,
                       Actuals := b,
                       Message := 'Arrays differ');

TEST_FINISHED();
END_METHOD

METHOD PRIVATE Test_DINT_Array_Equals
VAR
    a : ARRAY[2..7] OF DINT := [64, 98, 2147483647, -2147483648, 0, -63987538];
    b : ARRAY[2..7] OF DINT := [64, 98, 2147483647, -2147483648, 0, -63987538];
END_VAR
TEST('Test_DINT_Array_Equals');

AssertArrayEquals_DINT(Expecteds := a,
                       Actuals := b,
                       Message := 'Arrays differ');

TEST_FINISHED();
END_METHOD

METHOD PRIVATE Test_DWORD_Array_DifferInContent
VAR
    a : ARRAY[-2..1] OF DWORD := [16#6789ABCD, 16#EFAA2346, 16#ABABABAB, 16#EEEEEEEE];
    b : ARRAY[-2..1] OF DWORD := [16#6789ABCD, 16#EF012345, 16#ABABABAB, 16#EEEEEEEE];
END_VAR
TEST('Test_DWORD_Array_DifferInContent');

AssertArrayEquals_DWORD(Expecteds := a,
                        Actuals := b,
                        Message := 'Arrays differ');

TEST_FINISHED();
END_METHOD

METHOD PRIVATE Test_DWORD_Array_DifferInSize
VAR
    a : ARRAY[-2..1] OF DWORD := [16#6789ABCD, 16#EF012345, 16#67890ABC, 16#DDDDDDDD];
    b : ARRAY[-3..-2] OF DWORD := [16#6789ABCD, 16#EF012345];
END_VAR
TEST('Test_DWORD_Array_DifferInSize');

TCUNIT_ADSLOGSTR(msgCtrlMask := ADSLOG_MSGTYPE_ERROR,
                 msgFmtStr := 'This is just a string %s',
                 strArg := '10');

AssertArrayEquals_DWORD(Expecteds := a,
                        Actuals := b,
                        Message := 'Arrays differ');

TEST_FINISHED();
END_METHOD

METHOD PRIVATE Test_DWORD_Array_Equals
VAR
    a : ARRAY[2..3] OF DWORD := [16#6789ABCD, 16#EF012345];
    b : ARRAY[1..2] OF DWORD := [16#6789ABCD, 16#EF012345];
END_VAR
TEST('Test_DWORD_Array_Equals');

TCUNIT_ADSLOGSTR(msgCtrlMask := ADSLOG_MSGTYPE_ERROR,
                 msgFmtStr := 'This is just a string %s',
                 strArg := '9');

AssertArrayEquals_DWORD(Expecteds := a,
                        Actuals := b,
                        Message := 'Arrays differ');

TEST_FINISHED();
END_METHOD

METHOD PRIVATE Test_INT_Array_DifferInContent
VAR
    a : ARRAY[-8..-6] OF INT := [42, -23, -32768];
    b : ARRAY[1..3] OF INT := [42, 24, -32768];
END_VAR
TEST('Test_INT_Array_DifferInContent');

AssertArrayEquals_INT(Expecteds := a,
                      Actuals := b,
                      Message := 'Arrays differ');

TEST_FINISHED();
END_METHOD

METHOD PRIVATE Test_INT_Array_DifferInSize
VAR
    a : ARRAY[-4..3] OF INT := [64, 98, -32768, 32767, 5478, -378, 42, 6234];
    b : ARRAY[1..5] OF INT := [64, 98, -32768, 32767, 5478];
END_VAR
TEST('Test_INT_Array_DifferInSize');

AssertArrayEquals_INT(Expecteds := a,
                      Actuals := b,
                      Message := 'Arrays differ');

TEST_FINISHED();
END_METHOD

METHOD PRIVATE Test_INT_Array_Equals
VAR
    a : ARRAY[-5..1] OF INT := [64, 98, -32768, 32767, 5478, -378, 42];
    b : ARRAY[1..7] OF INT := [64, 98, -32768, 32767, 5478, -378, 42];
END_VAR
TEST('Test_INT_Array_Equals');

AssertArrayEquals_INT(Expecteds := a,
                      Actuals := b,
                      Message := 'Arrays differ');

TEST_FINISHED();
END_METHOD

METHOD PRIVATE Test_LINT_Array_DifferInContent
VAR
    a : ARRAY[-1..1] OF LINT := [9_223_372_036_854_775_807, -9_223_372_036_853_775_808, 55];
    b : ARRAY[4..6] OF LINT := [9_223_372_036_854_775_807, -9_223_372_036_854_775_808, 55];
END_VAR
TEST('Test_LINT_Array_DifferInContent');

AssertArrayEquals_LINT(Expecteds := a,
                       Actuals := b,
                       Message := 'Arrays differ');

TEST_FINISHED();
END_METHOD

METHOD PRIVATE Test_LINT_Array_DifferInSize
VAR
    a : ARRAY[-1..1] OF LINT := [9_223_372_036_854_775_807, -9_223_372_036_854_775_808, 55];
    b : ARRAY[4..5] OF LINT := [9_223_372_036_854_775_807, -9_223_372_036_854_775_808];
END_VAR
TEST('Test_LINT_Array_DifferInSize');

AssertArrayEquals_LINT(Expecteds := a,
                       Actuals := b,
                       Message := 'Arrays differ');

TEST_FINISHED();
END_METHOD

METHOD PRIVATE Test_LINT_Array_Equals
VAR
    a : ARRAY[-1..0] OF LINT := [9_223_372_036_854_775_807, -9_223_372_036_854_775_808];
    b : ARRAY[4..5] OF LINT := [9_223_372_036_854_775_807, -9_223_372_036_854_775_808];
END_VAR
TEST('Test_LINT_Array_Equals');

AssertArrayEquals_LINT(Expecteds := a,
                       Actuals := b,
                       Message := 'Arrays differ');

TEST_FINISHED();
END_METHOD

METHOD PRIVATE Test_LREAL_Array_DifferInContent
VAR
    a : ARRAY[-8..-6] OF LREAL := [42, -23, -32768];
    b : ARRAY[1..3] OF LREAL := [42, 24, -32768];
    c : ARRAY[-1..1] OF LREAL := [42, 0.0, -32768];
END_VAR
TEST('Test_LREAL_Array_DifferInContent');

AssertArrayEquals_LREAL(Expecteds := a,
                        Actuals := b,
                        Delta := 0.01,
                        Message := 'Arrays a and b differ');

MEMSET (ADR(c[0]), 255, SIZEOF(c[0]));

AssertArrayEquals_LREAL(Expecteds := a,
                        Actuals := c,
                        Delta := 0.01,
                        Message := 'Arrays a and c differ');

TEST_FINISHED();
END_METHOD

METHOD PRIVATE Test_LREAL_Array_DifferInSize
VAR
    a : ARRAY[-4..3] OF LREAL := [64, 98, -32768, 32767, 5478, -378, 42, 6234];
    b : ARRAY[1..5] OF LREAL := [64, 98, -32768, 32767, 5478];
END_VAR
TEST('Test_LREAL_Array_DifferInSize');

AssertArrayEquals_LREAL(Expecteds := a,
                        Actuals := b,
                        Delta := 0.01,
                        Message := 'Arrays differ');

TEST_FINISHED();
END_METHOD

METHOD PRIVATE Test_LREAL_Array_Equals
VAR
    a : ARRAY[-5..1] OF LREAL := [64.0, 98.1, -32768.2, 32767.3, 5478.4, -378.5, 42.6];
    b : ARRAY[1..7] OF LREAL := [64.0001, 98.0999, -32768.1995, 32767.3001, 5478.4002, -378.5003, 42.6001];
END_VAR
TEST('Test_LREAL_Array_Equals');

AssertArrayEquals_LREAL(Expecteds := a,
                        Actuals := b,
                        Delta := 0.01,
                        Message := 'Arrays differ');

TEST_FINISHED();
END_METHOD

METHOD PRIVATE Test_LREAL_Array2d_DifferInContent_LBOUND
VAR
    a : ARRAY[-5..-3,-1..1] OF LREAL := [      0,                        0.75069381424723836,      0.29093464244666262,     
                                               0.034287043863109802,     0.4487738206278411,       0.53067566153159162,      
                                               0.30748602156875937,      0.63373366540006071,      0.0090356068727726144 ];
                                                    
    b : ARRAY[0..2,3..5] OF LREAL :=   [       1,                        0.75069381424723836,      0.29093464244666262,     
                                               0.034287043883109802,     0.4487738206278411,       0.53067566153159162,      
                                               0.30748602156875937,      0.63373366540006071,      0.0090356068727726144 ];
END_VAR
TEST('Test_LREAL_Array2d_DifferInContent_LBOUND');

AssertArray2dEquals_LREAL(Expecteds := a,
                          Actuals := b,
                          Delta := 0.01,
                          Message := 'Arrays differ');

TEST_FINISHED();
END_METHOD

METHOD PRIVATE Test_LREAL_Array2d_DifferInContent_Middle
VAR
    a : ARRAY[-5..-3,-1..1] OF LREAL := [      0.39153705462419292,      0.75069381424723836,      0.29093464244666262,     
                                               0.034287043863109802,     0,                        0.53067566153159162,      
                                               0.30748602156875937,      0.63373366540006071,      0.0090356068727726144 ];
                                                    
    b : ARRAY[0..2,3..5] OF LREAL :=   [       0.39153705462419292,      0.75069381424723836,      0.29093464244666262,     
                                               0.034287043883109802,     1,                        0.53067566153159162,      
                                               0.30748602156875937,      0.63373366540006071,      0.0090356068727726144 ];
END_VAR
TEST('Test_LREAL_Array2d_DifferInContent_Middle');

AssertArray2dEquals_LREAL(Expecteds := a,
                          Actuals := b,
                          Delta := 0.01,
                          Message := 'Arrays differ');

TEST_FINISHED();
END_METHOD

METHOD PRIVATE Test_LREAL_Array2d_DifferInContent_UBOUND
VAR
    a : ARRAY[-5..-3,-1..1] OF LREAL := [      0.39153705462419292,      0.75069381424723836,      0.29093464244666262,     
                                               0.034287043863109802,     0.4487738206278411,       0.53067566153159162,      
                                               0.30748602156875937,      0.63373366540006071,      0                     ];
                                                    
    b : ARRAY[0..2,3..5] OF LREAL :=   [       0.39153705462419292,      0.75069381424723836,      0.29093464244666262,     
                                               0.034287043883109802,     0.4487738206278411,       0.53067566153159162,      
                                               0.30748602156875937,      0.63373366540006071,      1                     ];
END_VAR
TEST('Test_LREAL_Array2d_DifferInContent_UBOUND');

AssertArray2dEquals_LREAL(Expecteds := a,
                          Actuals := b,
                          Delta := 0.01,
                          Message := 'Arrays differ');

TEST_FINISHED();
END_METHOD

// Validate assertion for size difference in first dimension of 2d array
METHOD PRIVATE Test_LREAL_Array2d_DifferInSize_D1
VAR
    a : ARRAY[-4..-2, -1..0] OF LREAL := [    1.004110987573404E+62,  -2.873296335229452E+224,  
                                             -3.5901630626493139E+58, -1.0170839179102032E+220, 
                                             -1.1922268785979511E+79, -1.9309907712685427E+64    ];
                                           
    b : ARRAY[1..2, 0..1] OF LREAL := [       1.004110987573404E+62,  -2.873296335229452E+224,  
                                            -3.5901630626493139E+58,  -1.0170839179102032E+220   ];
END_VAR
TEST('Test_LREAL_Array2d_DifferInSize_D1');

AssertArray2dEquals_LREAL(Expecteds := a,
                          Actuals := b,
                          Delta := 0.01,
                          Message := 'Arrays differ');

TEST_FINISHED();
END_METHOD

// Validate assertion for size difference in second dimension of 2d array
METHOD PRIVATE Test_LREAL_Array2d_DifferInSize_D2
VAR
    a : ARRAY[-4..-3, -1..0] OF LREAL := [    1.004110987573404E+62,  -2.873296335229452E+224,  
                                             -3.5901630626493139E+58, -1.0170839179102032E+220    ];
                                           
    b : ARRAY[1..2, 0..2] OF LREAL :=    [    1.004110987573404E+62,  -2.873296335229452E+224,  -3.5901630626493139E+58,  
                                            -1.0170839179102032E+220,  -1.1922268785979511E+79,  -1.9309907712685427E+64  ];
END_VAR
TEST('Test_LREAL_Array2d_DifferInSize_D2');

AssertArray2dEquals_LREAL(Expecteds := a,
                          Actuals := b,
                          Delta := 0.01,
                          Message := 'Arrays differ');

TEST_FINISHED();
END_METHOD

METHOD PRIVATE Test_LREAL_Array2d_Equals
VAR
    a : ARRAY[-5..-3,-1..0] OF LREAL := [64.0, 98.1, -32768.2, 32767.3, 5478.4, -378.5];
    b : ARRAY[1..3,0..1] OF LREAL := [64.0001, 98.0999, -32768.1995, 32767.3001, 5478.4002, -378.5003];
END_VAR
TEST('Test_LREAL_Array2d_Equals');

AssertArray2dEquals_LREAL(Expecteds := a,
                          Actuals := b,
                          Delta := 0.01,
                          Message := 'Arrays differ');

TEST_FINISHED();
END_METHOD

METHOD PRIVATE Test_LREAL_Array3d_DifferInContent_LBOUND
VAR
    a : ARRAY[-5..-3,-1..1,1..3] OF LREAL := [      0,                        0.75069381424723836,      0.29093464244666262,     
                                                    0.034287043863109802,     0.4487738206278411,       0.53067566153159162,      
                                                    0.30748602156875937,      0.63373366540006071,      0.0090356068727726144,      

                                                    0.86311411432135576,      0.56920950420629679,      0.10704580466591092,
                                                    0.99235347099246152,      0.64118643600548919,      0.53803785449733854,
                                                    0.8536550946783531,       0.40930482857362593,      0.96201282039378433,

                                                    0.98258493467354446,      0.14997228521386732,      0.36854104388902942,
                                                    0.45163352808525487,      0.17645537628627167,      0.02055403311762681,
                                                    0.15098329919901829,      0.099172453907864375,     0.04804534513877954  ];
                                                    
    b : ARRAY[0..2,3..5,5..7] OF LREAL :=   [       1,                        0.75069381424723836,      0.29093464244666262,     
                                                    0.034287043883109802,     0.4487738206278411,       0.53067566153159162,      
                                                    0.30748602156875937,      0.63373366540006071,      0.0090356068727726144,      

                                                    0.86311411432135576,      0.56920950420629679,      0.10704582466591092,
                                                    0.99235347099246152,      0.64118643600548919,      0.53803785449733854,
                                                    0.8536556946783531,       0.40930482857362593,      0.96201282039378433,

                                                    0.98258493467354446,      0.14997228521386732,      0.36854104388952942,
                                                    0.45163352803525487,      0.17645537628627167,      0.02055403311762681,
                                                    0.15098329919901829,      0.099172453907864375,     0.04804534513877954  ];
END_VAR
TEST('Test_LREAL_Array3d_DifferInContent_LBOUND');

AssertArray3dEquals_LREAL(Expecteds := a,
                          Actuals := b,
                          Delta := 0.01,
                          Message := 'Arrays differ');

TEST_FINISHED();
END_METHOD

METHOD PRIVATE Test_LREAL_Array3d_DifferInContent_Middle
VAR
    a : ARRAY[-5..-3,-1..1,1..3] OF LREAL := [      0.39153705462419292,      0.75069381424723836,      0.29093464244666262,     
                                                    0.034287043863109802,     0.4487738206278411,       0.53067566153159162,      
                                                    0.30748602156875937,      0.63373366540006071,      0.0090356068727726144,      

                                                    0.86311411432135576,      0.56920950420629679,      0.10704580466591092,
                                                    0.99235347099246152,      0,                        0.53803785449733854,
                                                    0.8536550946783531,       0.40930482857362593,      0.96201282039378433,

                                                    0.98258493467354446,      0.14997228521386732,      0.36854104388902942,
                                                    0.45163352808525487,      0.17645537628627167,      0.02055403311762681,
                                                    0.15098329919901829,      0.099172453907864375,     0.04804534513877954  ];
                                                    
    b : ARRAY[0..2,3..5,5..7] OF LREAL :=   [       0.39153705462419292,      0.75069381424723836,      0.29093464244666262,     
                                                    0.034287043883109802,     0.4487738206278411,       0.53067566153159162,      
                                                    0.30748602156875937,      0.63373366540006071,      0.0090356068727726144,      

                                                    0.86311411432135576,      0.56920950420629679,      0.10704582466591092,
                                                    0.99235347099246152,      1,                        0.53803785449733854,
                                                    0.8536556946783531,       0.40930482857362593,      0.96201282039378433,

                                                    0.98258493467354446,      0.14997228521386732,      0.36854104388952942,
                                                    0.45163352803525487,      0.17645537628627167,      0.02055403311762681,
                                                    0.15098329919901829,      0.099172453907864375,     0.04804534513877954  ];
END_VAR
TEST('Test_LREAL_Array3d_DifferInContent_Middle');

AssertArray3dEquals_LREAL(Expecteds := a,
                          Actuals := b,
                          Delta := 0.01,
                          Message := 'Arrays differ');

TEST_FINISHED();
END_METHOD

METHOD PRIVATE Test_LREAL_Array3d_DifferInContent_UBOUND
VAR
    a : ARRAY[-5..-3,-1..1,1..3] OF LREAL := [      0.39153705462419292,      0.75069381424723836,      0.29093464244666262,     
                                                    0.034287043863109802,     0.4487738206278411,       0.53067566153159162,      
                                                    0.30748602156875937,      0.63373366540006071,      0.0090356068727726144,      

                                                    0.86311411432135576,      0.56920950420629679,      0.10704580466591092,
                                                    0.99235347099246152,      0.64118643600548919,      0.53803785449733854,
                                                    0.8536550946783531,       0.40930482857362593,      0.96201282039378433,

                                                    0.98258493467354446,      0.14997228521386732,      0.36854104388902942,
                                                    0.45163352808525487,      0.17645537628627167,      0.02055403311762681,
                                                    0.15098329919901829,      0.099172453907864375,     0                     ];
                                                    
    b : ARRAY[0..2,3..5,5..7] OF LREAL :=   [       0.39153705462419292,      0.75069381424723836,      0.29093464244666262,     
                                                    0.034287043883109802,     0.4487738206278411,       0.53067566153159162,      
                                                    0.30748602156875937,      0.63373366540006071,      0.0090356068727726144,      

                                                    0.86311411432135576,      0.56920950420629679,      0.10704582466591092,
                                                    0.99235347099246152,      0.64118643600548919,      0.53803785449733854,
                                                    0.8536556946783531,       0.40930482857362593,      0.96201282039378433,

                                                    0.98258493467354446,      0.14997228521386732,      0.36854104388952942,
                                                    0.45163352803525487,      0.17645537628627167,      0.02055403311762681,
                                                    0.15098329919901829,      0.099172453907864375,     1                     ];
END_VAR
TEST('Test_LREAL_Array3d_DifferInContent_UBOUND');

AssertArray3dEquals_LREAL(Expecteds := a,
                          Actuals := b,
                          Delta := 0.01,
                          Message := 'Arrays differ');

TEST_FINISHED();
END_METHOD

// Validate assertion for size difference in first dimension of 3d array
METHOD PRIVATE Test_LREAL_Array3d_DifferInSize_D1
VAR
    // 2x3x2
    a : ARRAY[-5..-4,0..2,-1..0] OF LREAL := [    2.082350040687358E+68,     1.0648482884583467E-159,  
                                                  2.6081154219341126E+236,  -2.2453945418753555E+134,  
                                                  8.5957093309297743E+301,  -5.9598471182139549E-139,  

                                                  -7.2419908660524697E+76,  5.0020389252645754E-160,  
                                                  -3.3631038290869421E-213,  -1.4376587532865779E+110,  
                                                  -1.0876803662003504E-263,  3.2352832374899203E+165  ];
    
    // 3x3x2
    b : ARRAY[0..2,3..5,6..7] OF LREAL := [    2.082350040687358E+68,     1.0648482884583467E-159,  
                                                  2.6081154219341126E+236,  -2.2453945418753555E+134,  
                                                  8.5957093309297743E+301,  -5.9598471182139549E-139,  

                                                  -7.2419908660524697E+76,  5.0020389252645754E-160,  
                                                  -3.3631038290869421E-213,  -1.4376587532865779E+110,  
                                                  -1.0876803662003504E-263,  3.2352832374899203E+165,

                                                  -4.6404382914454893E-67,  -1.3556949396573763E-104,  
                                                  -1.1830864377130754E+146,       7737.6071934405209,      
                                                  -470928678.08185887,       2.1842539859532993E-126    ];
END_VAR
TEST('Test_LREAL_Array3d_DifferInSize_D1');

AssertArray3dEquals_LREAL(Expecteds := a,
                          Actuals := b,
                          Delta := 0.01,
                          Message := 'Arrays differ');

TEST_FINISHED();
END_METHOD

// Validate assertion for size difference in second dimension of 3d array
METHOD PRIVATE Test_LREAL_Array3d_DifferInSize_D2
VAR
    // 2x3x2
    a : ARRAY[-5..-4,0..2,-1..0] OF LREAL := [    2.082350040687358E+68,     1.0648482884583467E-159,  
                                                  2.6081154219341126E+236,  -2.2453945418753555E+134,  
                                                  8.5957093309297743E+301,  -5.9598471182139549E-139,  

                                                  -7.2419908660524697E+76,  5.0020389252645754E-160,  
                                                  -3.3631038290869421E-213,  -1.4376587532865779E+110,  
                                                  -1.0876803662003504E-263,  3.2352832374899203E+165  ];
    
    // 2x2x2
    b : ARRAY[0..1,3..4,6..7] OF LREAL := [       2.082350040687358E+68,     1.0648482884583467E-159,  
                                                  2.6081154219341126E+236,  -2.2453945418753555E+134, 
 
                                                  8.5957093309297743E+301,  -5.9598471182139549E-139,  
                                                  -7.2419908660524697E+76,  5.0020389252645754E-160  ];
END_VAR
TEST('Test_LREAL_Array3d_DifferInSize_D2');

AssertArray3dEquals_LREAL(Expecteds := a,
                          Actuals := b,
                          Delta := 0.01,
                          Message := 'Arrays differ');

TEST_FINISHED();
END_METHOD

// Validate assertion for size difference in third dimension of 3d array
METHOD PRIVATE Test_LREAL_Array3d_DifferInSize_D3
VAR
    // 2x3x2
    a : ARRAY[-5..-4,0..2,-1..0] OF LREAL := [    2.082350040687358E+68,     1.0648482884583467E-159,  
                                                  2.6081154219341126E+236,  -2.2453945418753555E+134,  
                                                  8.5957093309297743E+301,  -5.9598471182139549E-139,  

                                                  -7.2419908660524697E+76,  5.0020389252645754E-160,  
                                                  -3.3631038290869421E-213,  -1.4376587532865779E+110,  
                                                  -1.0876803662003504E-263,  3.2352832374899203E+165  ];
    
    // 2x3x1
    b : ARRAY[0..1,3..5,6..6] OF LREAL := [       2.082350040687358E+68,     
                                                  1.0648482884583467E-159,  
                                                  2.6081154219341126E+236,  

                                                 -2.2453945418753555E+134,
                                                  8.5957093309297743E+301,  
                                                 -5.9598471182139549E-139  ];
END_VAR
TEST('Test_LREAL_Array3d_DifferInSize_D3');

AssertArray3dEquals_LREAL(Expecteds := a,
                          Actuals := b,
                          Delta := 0.01,
                          Message := 'Arrays differ');

TEST_FINISHED();
END_METHOD

METHOD PRIVATE Test_LREAL_Array3d_Equals
VAR
    a : ARRAY[-5..-4,-1..0,0..1] OF LREAL := [64.0, 98.1, -32768.2, 32767.3, 5478.4, -378.5, 42.6, 560344.0005];
    b : ARRAY[1..2,4..5,6..7] OF LREAL := [64.0001, 98.0999, -32768.1995, 32767.3001, 5478.4002, -378.5003, 42.6001, 560344.0006];
END_VAR
TEST('Test_LREAL_Array3d_Equals');

AssertArray3dEquals_LREAL(Expecteds := a,
                          Actuals := b,
                          Delta := 0.01,
                          Message := 'Arrays differ');

TEST_FINISHED();
END_METHOD

METHOD PRIVATE Test_LWORD_Array_DifferInContent
VAR
    a : ARRAY[1..1] OF LWORD := [16#EDCBA09876543210];
    b : ARRAY[1..1] OF LWORD := [16#01234567890ABCDE];
END_VAR
TEST('Test_LWORD_Array_DifferInContent');

AssertArrayEquals_LWORD(Expecteds := a,
                        Actuals := b,
                        Message := 'Arrays differ');

TEST_FINISHED();
END_METHOD

METHOD PRIVATE Test_LWORD_Array_DifferInSize
VAR
    a : ARRAY[1..1] OF LWORD := [16#EDCBA09876543210];
    b : ARRAY[1..2] OF LWORD := [16#01234567890ABCDE, 16#EDCBA09876543210];
END_VAR
TEST('Test_LWORD_Array_DifferInSize');

AssertArrayEquals_LWORD(Expecteds := a,
                        Actuals := b,
                        Message := 'Arrays differ');

TEST_FINISHED();
END_METHOD

METHOD PRIVATE Test_LWORD_Array_Equals
VAR
    a : ARRAY[1..2] OF LWORD := [16#01234567890ABCDE, 16#EDCBA09876543210];
    b : ARRAY[1..2] OF LWORD := [16#01234567890ABCDE, 16#EDCBA09876543210];
END_VAR
TEST('Test_LWORD_Array_Equals');

AssertArrayEquals_LWORD(Expecteds := a,
                        Actuals := b,
                        Message := 'Arrays differ');

TEST_FINISHED();
END_METHOD

METHOD PRIVATE Test_REAL_Array_DifferInContent
VAR
    a : ARRAY[-8..-6] OF REAL := [42, -23, -32768];
    b : ARRAY[1..3] OF REAL := [42, 24, -32768];
    c : ARRAY[-1..1] OF REAL := [42, 0.0, -32768];
END_VAR
TEST('Test_REAL_Array_DifferInContent');

AssertArrayEquals_REAL(Expecteds := a,
                       Actuals := b,
                       Delta := 0.01,
                       Message := 'Arrays a and b differ');

MEMSET (ADR(c[0]), 255, SIZEOF(c[0]));

AssertArrayEquals_REAL(Expecteds := a,
                       Actuals := c,
                       Delta := 0.01,
                       Message := 'Arrays a and c differ');

TEST_FINISHED();
END_METHOD

METHOD PRIVATE Test_REAL_Array_DifferInSize
VAR
    a : ARRAY[-4..3] OF REAL := [64, 98, -32768, 32767, 5478, -378, 42, 6234];
    b : ARRAY[1..5] OF REAL := [64, 98, -32768, 32767, 5478];
END_VAR
TEST('Test_REAL_Array_DifferInSize');

TCUNIT_ADSLOGSTR(msgCtrlMask := ADSLOG_MSGTYPE_WARN,
                 msgFmtStr := 'This is just a string %s',
                 strArg := '12');

AssertArrayEquals_REAL(Expecteds := a,
                       Actuals := b,
                       Delta := 0.01,
                       Message := 'Arrays differ');

TEST_FINISHED();
END_METHOD

METHOD PRIVATE Test_REAL_Array_Equals
VAR
    a : ARRAY[-5..1] OF REAL := [64.0, 98.1, -32768.2, 32767.3, 5478.4, -378.5, 42.6];
    b : ARRAY[1..7] OF REAL := [64.0001, 98.0999, -32768.1995, 32767.3001, 5478.4002, -378.5003, 42.6001];
END_VAR
TEST('Test_REAL_Array_Equals');

TCUNIT_ADSLOGSTR(msgCtrlMask := ADSLOG_MSGTYPE_WARN,
                 msgFmtStr := 'This is just a string %s',
                 strArg := '11');

AssertArrayEquals_REAL(Expecteds := a,
                       Actuals := b,
                       Delta := 0.01,
                       Message := 'Arrays differ');

TEST_FINISHED();
END_METHOD

METHOD PRIVATE Test_REAL_Array2d_DifferInContent_LBOUND
VAR
    a : ARRAY[-5..-3,-1..1] OF REAL := [      0,                0.349414557,      0.806114793,      
                                              0.832643092,      0.676487744,      0.422208548,       
                                               0.58663553,      0.108467624,      0.153285101  ];
                                               
    b : ARRAY[1..3,0..2] OF REAL :=    [      1,               0.349414557,      0.80611479,      
                                              0.83264309,      0.67648774,      0.42220855,       
                                               0.5866355,      0.108467624,      0.153285101  ];
END_VAR
TEST('Test_REAL_Array2d_DifferInContent_LBOUND');

AssertArray2dEquals_REAL(Expecteds := a,
                         Actuals := b,
                         Delta := 0.01,
                         Message := 'Arrays differ');

TEST_FINISHED();
END_METHOD

METHOD PRIVATE Test_REAL_Array2d_DifferInContent_Middle
VAR
    a : ARRAY[-5..-3,-1..1] OF REAL := [      0.555157363,      0.349414557,      0.806114793,      
                                              0.832643092,      0,                0.422208548,       
                                               0.58663553,      0.108467624,      0.153285101  ];
                                               
    b : ARRAY[1..3,0..2] OF REAL :=    [      0.555157363,      0.349414557,      0.80611479,      
                                              0.83264309,      1,                 0.42220855,       
                                               0.5866355,      0.108467624,       0.153285101  ];
END_VAR
TEST('Test_REAL_Array2d_DifferInContent_Middle');

AssertArray2dEquals_REAL(Expecteds := a,
                         Actuals := b,
                         Delta := 0.01,
                         Message := 'Arrays differ');

TEST_FINISHED();
END_METHOD

METHOD PRIVATE Test_REAL_Array2d_DifferInContent_UBOUND
VAR
    a : ARRAY[-5..-3,-1..1] OF REAL := [      0.555157363,      0.349414557,      0.806114793,      
                                              0.832643092,      0.676487744,      0.422208548,       
                                               0.58663553,      0.108467624,      0           ];
                                               
    b : ARRAY[1..3,0..2] OF REAL :=    [      0.555157363,      0.349414557,      0.80611479,      
                                              0.83264309,      0.67648774,      0.42220855,       
                                               0.5866355,      0.108467624,      1            ];
END_VAR
TEST('Test_REAL_Array2d_DifferInContent_UBOUND');

AssertArray2dEquals_REAL(Expecteds := a,
                         Actuals := b,
                         Delta := 0.01,
                         Message := 'Arrays differ');

TEST_FINISHED();
END_METHOD

// Validate assertion for size difference in first dimension of 2d array
METHOD PRIVATE Test_REAL_Array2d_DifferInSize_D1
VAR
    a : ARRAY[-4..-2, -1..0] OF REAL := [   6.89723951E-35, 1.255877E-08,   
                                            1.31490056E+30, 1.0130173,
                                            7.50187543E-38, -698122.938  ];
                                           
    b : ARRAY[1..2, 0..1] OF REAL :=    [   6.89723951E-35, 1.255877E-08,   
                                            1.31490056E+30, 1.0130173   ];
END_VAR
TEST('Test_REAL_Array2d_DifferInSize_D1');

AssertArray2dEquals_REAL(Expecteds := a,
                         Actuals := b,
                         Delta := 0.01,
                         Message := 'Arrays differ');

TEST_FINISHED();
END_METHOD

// Validate assertion for size difference in second dimension of 2d array
METHOD PRIVATE Test_REAL_Array2d_DifferInSize_D2
VAR
    a : ARRAY[-4..-3, -1..0] OF REAL := [   6.89723951E-35, 1.255877E-08,
                                            1.31490056E+30, 1.0130173   ];
                                           
    b : ARRAY[1..2, 0..2] OF REAL :=    [   6.89723951E-35, 1.255877E-08,   1.31490056E+30,
                                            1.0130173,      7.50187543E-38,   -698122.938  ];
END_VAR
TEST('Test_REAL_Array2d_DifferInSize_D2');

AssertArray2dEquals_REAL(Expecteds := a,
                         Actuals := b,
                         Delta := 0.01,
                         Message := 'Arrays differ');

TEST_FINISHED();
END_METHOD

METHOD PRIVATE Test_REAL_Array2d_Equals
VAR
    a : ARRAY[-5..-3,-1..0] OF REAL := [64.0, 98.1, -32768.2, 32767.3, 5478.4, -378.5];
    b : ARRAY[1..3,0..1] OF REAL := [64.0001, 98.0999, -32768.1995, 32767.3001, 5478.4002, -378.5003];
END_VAR
TEST('Test_REAL_Array2d_Equals');

AssertArray2dEquals_REAL(Expecteds := a,
                         Actuals := b,
                         Delta := 0.01,
                         Message := 'Arrays differ');

TEST_FINISHED();
END_METHOD

METHOD PRIVATE Test_REAL_Array3d_DifferInContent_LBOUND
VAR
    a : ARRAY[-5..-3,-1..1,0..2] OF REAL := [       0,                0.349414557,     0.806114793,      
                                                    0.832643092,      0.676487744,     0.422208548,       
                                                    0.58663553,       0.108467624,     0.153285101,      

                                                    0.331847638,      0.518251598,     0.396329135,       
                                                    0.68058759,       0.837357402,     0.0384598672,      
                                                    0.485841662,      0.103918776,     0.662022889,      

                                                    0.576529145,      0.341899037,     0.375482976,       
                                                    0.77158308,       0.64138025,      0.780365825,      
                                                    0.680897593,      0.451427311,     0.151570886  ];
                                                    
    b : ARRAY[1..3,3..5,6..8] OF REAL :=    [       1,                0.349414557,     0.806116793,      
                                                    0.832643092,      0.676487744,     0.422208548,       
                                                    0.58663553,       0.108467624,     0.153285101,      

                                                    0.331847638,      0.518251598,     0.396329135,       
                                                    0.68058759,       0.837357402,     0.0384598672,      
                                                    0.485844662,      0.103918776,     0.662022889,      

                                                    0.576529145,      0.341899037,     0.375482976,       
                                                    0.77158308,       0.64138125,      0.780365825,      
                                                    0.680897593,      0.451427311,     0.151520886  ];
END_VAR
TEST('Test_REAL_Array3d_DifferInContent_LBOUND');

AssertArray3dEquals_REAL(Expecteds := a,
                         Actuals := b,
                         Delta := 0.01,
                         Message := 'Arrays differ');

TEST_FINISHED();
END_METHOD

METHOD PRIVATE Test_REAL_Array3d_DifferInContent_Middle
VAR
    a : ARRAY[-5..-3,-1..1,0..2] OF REAL := [       0.555157363,      0.349414557,     0.806114793,      
                                                    0.832643092,      0.676487744,     0.422208548,       
                                                    0.58663553,       0.108467624,     0.153285101,      

                                                    0.331847638,      0.518251598,     0.396329135,       
                                                    0.68058759,       0,               0.0384598672,      
                                                    0.485841662,      0.103918776,     0.662022889,      

                                                    0.576529145,      0.341899037,     0.375482976,       
                                                    0.77158308,       0.64138025,      0.780365825,      
                                                    0.680897593,      0.451427311,     0.151570886  ];
                                                    
    b : ARRAY[1..3,3..5,6..8] OF REAL :=    [       0.555157363,      0.349414557,     0.806116793,      
                                                    0.832643092,      0.676487744,     0.422208548,       
                                                    0.58663553,       0.108467624,     0.153285101,      

                                                    0.331847638,      0.518251598,     0.396329135,       
                                                    0.68058759,       1,               0.0384598672,      
                                                    0.485844662,      0.103918776,     0.662022889,      

                                                    0.576529145,      0.341899037,     0.375482976,       
                                                    0.77158308,       0.64138125,      0.780365825,      
                                                    0.680897593,      0.451427311,     0.151520886  ];
END_VAR
TEST('Test_REAL_Array3d_DifferInContent_Middle');

AssertArray3dEquals_REAL(Expecteds := a,
                         Actuals := b,
                         Delta := 0.01,
                         Message := 'Arrays differ');

TEST_FINISHED();
END_METHOD

METHOD PRIVATE Test_REAL_Array3d_DifferInContent_UBOUND
VAR
    a : ARRAY[-5..-3,-1..1,0..2] OF REAL := [       0.555157363,      0.349414557,     0.806114793,      
                                                    0.832643092,      0.676487744,     0.422208548,       
                                                    0.58663553,       0.108467624,     0.153285101,      

                                                    0.331847638,      0.518251598,     0.396329135,       
                                                    0.68058759,       0.837357402,     0.0384598672,      
                                                    0.485841662,      0.103918776,     0.662022889,      

                                                    0.576529145,      0.341899037,     0.375482976,       
                                                    0.77158308,       0.64138025,      0.780365825,      
                                                    0.680897593,      0.451427311,     0              ];
                                                    
    b : ARRAY[1..3,3..5,6..8] OF REAL :=    [       0.555157363,      0.349414557,     0.806116793,      
                                                    0.832643092,      0.676487744,     0.422208548,       
                                                    0.58663553,       0.108467624,     0.153285101,      

                                                    0.331847638,      0.518251598,     0.396329135,       
                                                    0.68058759,       0.837357402,     0.0384598672,      
                                                    0.485844662,      0.103918776,     0.662022889,      

                                                    0.576529145,      0.341899037,     0.375482976,       
                                                    0.77158308,       0.64138125,      0.780365825,      
                                                    0.680897593,      0.451427311,     1              ];
END_VAR
TEST('Test_REAL_Array3d_DifferInContent_UBOUND');

AssertArray3dEquals_REAL(Expecteds := a,
                         Actuals := b,
                         Delta := 0.01,
                         Message := 'Arrays differ');

TEST_FINISHED();
END_METHOD

// Validate assertion for size difference in first dimension of 3d array
METHOD PRIVATE Test_REAL_Array3d_DifferInSize_D1
VAR
    // 2x3x2
    a : ARRAY[-5..-4,1..3,-2..-1] OF REAL := [   4.10516757E-36,        666455872,  
                                                 -6.32274414E-23,   2.51930489E-20,      
                                                -13.6131887,        6.56142373E+29,   

                                                 -7.4229119E+36,   -1.19216618E+17,  
                                                 -1.76541143E+10,   1.06367558E+38,   
                                                  9.62853863E+24,  -1.02125985E-17  ];
                                                  
    // 1x3x2                                      
    b : ARRAY[1..1,4..6,6..7] OF REAL :=  [   4.10516757E-36,        666455872,  
                                                 -6.32274414E-23,   2.51930489E-20,      
                                                -13.6131887,        6.56142373E+29 ];
END_VAR
TEST('Test_REAL_Array3d_DifferInSize_D1');

AssertArray3dEquals_REAL(Expecteds := a,
                         Actuals := b,
                         Delta := 0.01,
                         Message := 'Arrays differ');

TEST_FINISHED();
END_METHOD

// Validate assertion for size difference in second dimension of 3d array
METHOD PRIVATE Test_REAL_Array3d_DifferInSize_D2
VAR
    // 2x3x2
    a : ARRAY[-5..-4,1..3,-2..-1] OF REAL := [   4.10516757E-36,        666455872,  
                                                 -6.32274414E-23,   2.51930489E-20,      
                                                -13.6131887,        6.56142373E+29,   

                                                 -7.4229119E+36,   -1.19216618E+17,  
                                                 -1.76541143E+10,   1.06367558E+38,   
                                                  9.62853863E+24,  -1.02125985E-17  ];

    // 2x2x2                                      
    b : ARRAY[1..2,4..5,6..7] OF REAL :=  [       4.10516757E-36,        666455872,  
                                                 -6.32274414E-23,   2.51930489E-20,      

                                                -13.6131887,        6.56142373E+29,   
                                                 -7.4229119E+36,   -1.19216618E+17  ];
END_VAR
TEST('Test_REAL_Array3d_DifferInSize_D2');

AssertArray3dEquals_REAL(Expecteds := a,
                         Actuals := b,
                         Delta := 0.01,
                         Message := 'Arrays differ');

TEST_FINISHED();
END_METHOD

// Validate assertion for size difference in third dimension of 3d array
METHOD PRIVATE Test_REAL_Array3d_DifferInSize_D3
VAR
    // 2x3x2
    a : ARRAY[-5..-4,1..3,-2..-1] OF REAL := [   4.10516757E-36,        666455872,  
                                                 -6.32274414E-23,   2.51930489E-20,      
                                                -13.6131887,        6.56142373E+29,   

                                                 -7.4229119E+36,   -1.19216618E+17,  
                                                 -1.76541143E+10,   1.06367558E+38,   
                                                  9.62853863E+24,  -1.02125985E-17  ];
                                                  
    // 2x3x1
    b : ARRAY[1..2,4..6,6..6] OF REAL :=  [       4.10516757E-36,        
                                                        666455872,  
                                                  -6.32274414E-23,
   
                                                  2.51930489E-20,      
                                                     -13.6131887,   
                                                  6.56142373E+29 ]; 
END_VAR
TEST('Test_REAL_Array3d_DifferInSize_D3');

AssertArray3dEquals_REAL(Expecteds := a,
                         Actuals := b,
                         Delta := 0.01,
                         Message := 'Arrays differ');

TEST_FINISHED();
END_METHOD

METHOD PRIVATE Test_REAL_Array3d_Equals
VAR
    a : ARRAY[-5..-4,-1..0,0..1] OF REAL := [64.0, 98.1, -32768.2, 32767.3, 5478.4, -378.5, 42.6, 560344.0005];
    b : ARRAY[1..2,4..5,6..7] OF REAL := [64.0001, 98.0999, -32768.1995, 32767.3001, 5478.4002, -378.5003, 42.6001, 560344.0006];
END_VAR
TEST('Test_REAL_Array3d_Equals');

AssertArray3dEquals_REAL(Expecteds := a,
                         Actuals := b,
                         Delta := 0.01,
                         Message := 'Arrays differ');

TEST_FINISHED();
END_METHOD

METHOD PRIVATE Test_SINT_Array_DifferInContent
VAR
    a : ARRAY[0..0] OF SINT := [-128];
    b : ARRAY[0..0] OF SINT := [127];
END_VAR
TEST('Test_SINT_Array_DifferInContent');

AssertArrayEquals_SINT(Expecteds := a,
                       Actuals := b,
                       Message := 'Arrays differ');

TEST_FINISHED();
END_METHOD

METHOD PRIVATE Test_SINT_Array_DifferInSize
VAR
    a : ARRAY[0..0] OF SINT := [-128];
    b : ARRAY[0..1] OF SINT := [-128, 127];
END_VAR
TEST('Test_SINT_Array_DifferInSize');

AssertArrayEquals_SINT(Expecteds := a,
                       Actuals := b,
                       Message := 'Arrays differ');

TEST_FINISHED();
END_METHOD

METHOD PRIVATE Test_SINT_Array_Equals
VAR
    a : ARRAY[0..3] OF SINT := [-128, 127, -34, 62];
    b : ARRAY[0..3] OF SINT := [-128, 127, -34, 62];
END_VAR
TEST('Test_SINT_Array_Equals');

AssertArrayEquals_SINT(Expecteds := a,
                       Actuals := b,
                       Message := 'Arrays differ');

TEST_FINISHED();
END_METHOD

METHOD PRIVATE Test_UDINT_Array_DifferInContent
VAR
    a : ARRAY[-5..-4] OF UDINT := [4294967295, 5];
    b : ARRAY[0..1] OF UDINT := [4294967295, 4];
END_VAR
TEST('Test_UDINT_Array_DifferInContent');

AssertArrayEquals_UDINT(Expecteds := a,
                        Actuals := b,
                        Message := 'Arrays differ');

TEST_FINISHED();
END_METHOD

METHOD PRIVATE Test_UDINT_Array_DifferInSize
VAR
    a : ARRAY[-5..-4] OF UDINT := [4294967295, 0];
    b : ARRAY[0..2] OF UDINT := [4294967295, 0, 5000];
END_VAR
TEST('Test_UDINT_Array_DifferInSize');

AssertArrayEquals_UDINT(Expecteds := a,
                        Actuals := b,
                        Message := 'Arrays differ');

TEST_FINISHED();
END_METHOD

METHOD PRIVATE Test_UDINT_Array_Equals
VAR
    a : ARRAY[1..3] OF UDINT := [0, 4294967295, 5000];
    b : ARRAY[1..3] OF UDINT := [0, 4294967295, 5000];
END_VAR
TEST('Test_UDINT_Array_Equals');

AssertArrayEquals_UDINT(Expecteds := a,
                        Actuals := b,
                        Message := 'Arrays differ');

TEST_FINISHED();
END_METHOD

METHOD PRIVATE Test_UINT_Array_DifferInContent
VAR
    a : ARRAY[0..3] OF UINT := [0, 4, 8, 99];
    b : ARRAY[0..3] OF UINT := [0, 4, 8, 12];
END_VAR
TEST('Test_UINT_Array_DifferInContent');

AssertArrayEquals_UINT(Expecteds := a,
                       Actuals := b,
                       Message := 'Arrays differ');

TEST_FINISHED();
END_METHOD

METHOD PRIVATE Test_UINT_Array_DifferInSize
VAR
    a : ARRAY[0..2] OF UINT := [0, 4, 8];
    b : ARRAY[0..3] OF UINT := [0, 4, 8, 12];
END_VAR
TEST('Test_UINT_Array_DifferInSize');

AssertArrayEquals_UINT(Expecteds := a,
                       Actuals := b,
                       Message := 'Arrays differ');

TEST_FINISHED();
END_METHOD

METHOD PRIVATE Test_UINT_Array_Equals
VAR
    a : ARRAY[0..4] OF UINT := [0, 65535, 2000, 34123, 59];
    b : ARRAY[0..4] OF UINT := [0, 65535, 2000, 34123, 59];
END_VAR
TEST('Test_UINT_Array_Equals');

AssertArrayEquals_UINT(Expecteds := a,
                       Actuals := b,
                       Message := 'Arrays differ');

TEST_FINISHED();
END_METHOD

METHOD PRIVATE Test_ULINT_Array_DifferInContent
VAR
    a : ARRAY[0..1] OF ULINT := [3_213_000_444_000, 9_400_000_000_000];
    b : ARRAY[0..1] OF ULINT := [3_213_000_444_000, 18_446_744_073_709_551_615];
END_VAR
TEST('Test_ULINT_Array_DifferInContent');

AssertArrayEquals_ULINT(Expecteds := a,
                        Actuals := b,
                        Message := 'Arrays differ');

TEST_FINISHED();
END_METHOD

METHOD PRIVATE Test_ULINT_Array_DifferInSize
VAR
    a : ARRAY[0..1] OF ULINT := [0, 9_400_000_000_000];
    b : ARRAY[0..0] OF ULINT := [0];
END_VAR
TEST('Test_ULINT_Array_DifferInSize');

AssertArrayEquals_ULINT(Expecteds := a,
                        Actuals := b,
                        Message := 'Arrays differ');

TEST_FINISHED();
END_METHOD

METHOD PRIVATE Test_ULINT_Array_Equals
VAR
    a : ARRAY[0..3] OF ULINT := [0, 18_446_744_073_709_551_615, 9_400_000_000_000, 3_213_000_444_000];
    b : ARRAY[0..3] OF ULINT := [0, 18_446_744_073_709_551_615, 9_400_000_000_000, 3_213_000_444_000];
END_VAR
TEST('Test_ULINT_Array_Equals');

AssertArrayEquals_ULINT(Expecteds := a,
                        Actuals := b,
                        Message := 'Arrays differ');

TEST_FINISHED();
END_METHOD

METHOD PRIVATE Test_USINT_Array_DifferInContent
VAR
    a : ARRAY[0..10] OF USINT := [0,1,2,3,6(4),5];
    b : ARRAY[0..10] OF USINT := [0,1,2,3,6(5),6];
END_VAR
TEST('Test_USINT_Array_DifferInContent');

AssertArrayEquals_USINT(Expecteds := a,
                        Actuals := b,
                        Message := 'Arrays differ');

TEST_FINISHED();
END_METHOD

METHOD PRIVATE Test_USINT_Array_DifferInSize
VAR
    a : ARRAY[0..100] OF USINT := [101(42)];
    b : ARRAY[0..70] OF USINT := [71(42)];
END_VAR
TEST('Test_USINT_Array_DifferInSize');

AssertArrayEquals_USINT(Expecteds := a,
                        Actuals := b,
                        Message := 'Arrays differ');

TEST_FINISHED();
END_METHOD

METHOD PRIVATE Test_USINT_Array_Equals
VAR
    a : ARRAY[0..100] OF USINT := [42, 100(33)];
    b : ARRAY[0..100] OF USINT := [42, 100(33)];
END_VAR
TEST('Test_USINT_Array_Equals');

AssertArrayEquals_USINT(Expecteds := a,
                        Actuals := b,
                        Message := 'Arrays differ');

TEST_FINISHED();
END_METHOD

METHOD PRIVATE Test_WORD_Array_DifferInContent
VAR
    a : ARRAY[1..7] OF WORD := [16#2323, 16#876A, 16#4CD4, 16#F3DC, 16#BBBB, 16#FFFF, 16#1133];
    b : ARRAY[1..7] OF WORD := [16#2323, 16#876A, 16#4CD4, 16#F3DC, 16#BBBB, 16#FFFF, 16#1122];
END_VAR
TEST('Test_WORD_Array_DifferInContent');

AssertArrayEquals_WORD(Expecteds := a,
                       Actuals := b,
                       Message := 'Arrays differ');

TEST_FINISHED();
END_METHOD

METHOD PRIVATE Test_WORD_Array_DifferInSize
VAR
    a : ARRAY[1..5] OF WORD := [16#0000, 16#3333, 16#5555, 16#7777, 16#BBBB];
    b : ARRAY[1..7] OF WORD := [16#0000, 16#3333, 16#5555, 16#7777, 16#BBBB, 16#FFFF, 16#1122];
END_VAR
TEST('Test_WORD_Array_DifferInSize');

AssertArrayEquals_WORD(Expecteds := a,
                       Actuals := b,
                       Message := 'Arrays differ');

TEST_FINISHED();
END_METHOD

METHOD PRIVATE Test_WORD_Array_Equals
VAR
    a : ARRAY[1..5] OF WORD := [16#AAAA, 16#BBBB, 16#CCCC, 16#DDDD, 16#EEEE];
    b : ARRAY[1..5] OF WORD := [16#AAAA, 16#BBBB, 16#CCCC, 16#DDDD, 16#EEEE];
END_VAR
TEST('Test_WORD_Array_Equals');

AssertArrayEquals_WORD(Expecteds := a,
                       Actuals := b,
                       Message := 'Arrays differ');

TEST_FINISHED();
END_METHOD

END_FUNCTION_BLOCK

// ---- Test/FB_CreateDisabledTest.TcPOU
(*
    This testsuite runs two tests. One that is enabled (and that is supposed to fail), and one that is disabled (and
    even though it also is failing is not supposed to run).
*)
FUNCTION_BLOCK FB_CreateDisabledTest EXTENDS TcUnit.FB_TestSuite

TestEnabled();
TestDisabled();

METHOD PRIVATE TestDisabled
VAR
    a : BOOL := FALSE;
    b : BOOL := TRUE;
END_VAR
TEST('DISABLED_ThisShouldNotExecute');

AssertEquals(Expected := a,
             Actual := b,
             Message := 'A does not equal B');

TEST_FINISHED();
END_METHOD

METHOD PRIVATE TestEnabled
VAR
    a : BOOL := TRUE;
    b : BOOL := FALSE;
END_VAR
TEST('TestEnabled');

AssertEquals(Expected := a,
             Actual := b,
             Message := 'A does not equal B');

TEST_FINISHED();
END_METHOD

END_FUNCTION_BLOCK

// ---- Test/FB_AnyPrimitiveTypes.TcPOU
(*
    This testsuite tests the different assert-functions for all the primitive data types in TwinCAT, but using the
    ANY-version of the Assert-method.
    For every data type at least two different tests have been defined:
        1. One test that succeeds (Expected and actual are equal)
        2. One test that fails (Expected and actual are false).
    For every failing test the printed value should be the same as if we were using the primitive data type assert
    directly. 
*)
FUNCTION_BLOCK FB_AnyPrimitiveTypes EXTENDS TcUnit.FB_TestSuite

Test_ANY_BYTE_Equals();
Test_ANY_BYTE_Differ();
Test_ANY_BOOL_Equals();
Test_ANY_BOOL_Differ();
Test_ANY_DATE_Equals();
Test_ANY_DATE_Differ();
Test_ANY_DATE_AND_TIME_Equals();
Test_ANY_DATE_AND_TIME_Differ();
Test_ANY_DINT_Equals();
Test_ANY_DINT_Differ();
Test_ANY_DWORD_Equals();
Test_ANY_DWORD_Differ();
Test_ANY_INT_Equals();
Test_ANY_INT_Differ();
Test_ANY_LINT_Equals();
Test_ANY_LINT_Differ();
Test_ANY_LREAL_Equals();
Test_ANY_LREAL_Differ();
Test_ANY_LTIME_Equals();
Test_ANY_LTIME_Differ();
Test_ANY_LWORD_Equals();
Test_ANY_LWORD_Differ();
Test_ANY_REAL_Equals();
Test_ANY_REAL_Differ();
Test_ANY_SINT_Equals();
Test_ANY_SINT_Differ();
Test_ANY_STRING_Equals();
Test_ANY_STRING_Differ();
Test_ANY_STRING_Differ_2();
Test_ANY_TIME_Equals();
Test_ANY_TIME_Differ();
Test_ANY_TIME_OF_DAY_Equals();
TesT_ANY_TIME_OF_DAY_Differ();
Test_ANY_UDINT_Equals();
Test_ANY_UDINT_Differ();
Test_ANY_UINT_Equals();
Test_ANY_UINT_Differ();
Test_ANY_ULINT_Equals();
Test_ANY_ULINT_Differ();
Test_ANY_USINT_Equals();
Test_ANY_USINT_Differ();
Test_ANY_WORD_Equals();
Test_ANY_WORD_Differ();
Test_ANY_WSTRING_Equals();
Test_ANY_WSTRING_Differ();
Test_ANY_WSTRING_Differ_2();

METHOD PRIVATE Test_ANY_BOOL_Differ
VAR
    a : BOOL := TRUE;
    b : BOOL := FALSE;
END_VAR
TEST('Test_ANY_BOOL_Differ');

AssertEquals(Expected := a,
             Actual := b,
             Message := 'Values differ');

TEST_FINISHED();
END_METHOD

METHOD PRIVATE Test_ANY_BOOL_Equals
VAR
    a : BOOL := TRUE;
    b : BOOL := TRUE;
END_VAR
TEST('Test_ANY_BOOL_Equals');

AssertEquals(Expected := a,
             Actual := b,
             Message := 'Values differ');

TEST_FINISHED();
END_METHOD

METHOD PRIVATE Test_ANY_BYTE_Differ
VAR
    a : BYTE := 16#AB;
    b : BYTE := 16#CD;
END_VAR
TEST('Test_ANY_BYTE_Differ');

AssertEquals(Expected := a,
             Actual := b,
             Message := 'Values differ');

TEST_FINISHED();
END_METHOD

METHOD PRIVATE Test_ANY_BYTE_Equals
VAR
    a : BYTE := 16#CD;
    b : BYTE := 16#CD;
END_VAR
TEST('Test_ANY_BYTE_Equals');

AssertEquals(Expected := a,
             Actual := b,
             Message := 'Values differ');

TEST_FINISHED();
END_METHOD

METHOD PRIVATE Test_ANY_DATE_AND_TIME_Differ
VAR
    a : DATE_AND_TIME := DATE_AND_TIME#1996-05-06-15:36:30;
    b : DATE_AND_TIME := DATE_AND_TIME#1972-03-29-00:00:00;
END_VAR
TEST('Test_ANY_DATE_AND_TIME_Differ');

AssertEquals(Expected := a,
             Actual := b,
             Message := 'Values differ');

TEST_FINISHED();
END_METHOD

METHOD PRIVATE Test_ANY_DATE_AND_TIME_Equals
VAR
    a : DATE_AND_TIME := DATE_AND_TIME#2019-01-20-13:54:30;
    b : DATE_AND_TIME := DATE_AND_TIME#2019-01-20-13:54:30;
END_VAR
TEST('Test_ANY_DATE_AND_TIME_Equals');

AssertEquals(Expected := a,
             Actual := b,
             Message := 'Values differ');

TEST_FINISHED();
END_METHOD

METHOD PRIVATE Test_ANY_DATE_Differ
VAR
    a : DATE := DATE#1996-05-06;
    b : DATE := DATE#2019-01-20;
END_VAR
TEST('Test_ANY_DATE_Differ');

AssertEquals(Expected := a,
             Actual := b,
             Message := 'Values differ');

TEST_FINISHED();
END_METHOD

METHOD PRIVATE Test_ANY_DATE_Equals
VAR
    a : DATE := DATE#1996-05-06;
    b : DATE := DATE#1996-05-06;
END_VAR
TEST('Test_ANY_DATE_Equals');

AssertEquals(Expected := a,
             Actual := b,
             Message := 'Values differ');

TEST_FINISHED();
END_METHOD

METHOD PRIVATE Test_ANY_DINT_Differ
VAR
    a : DINT := -55555;
    b : DINT := 70000;
END_VAR
TEST('Test_ANY_DINT_Differ');

AssertEquals(Expected := a,
             Actual := b,
             Message := 'Values differ');

TEST_FINISHED();
END_METHOD

METHOD PRIVATE Test_ANY_DINT_Equals
VAR
    a : DINT := -80000;
    b : DINT := -80000;
END_VAR
TEST('Test_ANY_DINT_Equals');

AssertEquals(Expected := a,
             Actual := b,
             Message := 'Values differ');

TEST_FINISHED();
END_METHOD

METHOD PRIVATE Test_ANY_DWORD_Differ
VAR
    a : DWORD := 16#12345678;
    b : DWORD := 16#90ABCDEF;
END_VAR
TEST('Test_ANY_DWORD_Differ');

AssertEquals(Expected := a,
             Actual := b,
             Message := 'Values differ');

TEST_FINISHED();
END_METHOD

METHOD PRIVATE Test_ANY_DWORD_Equals
VAR
    a : DWORD := 16#7890ABCD;
    b : DWORD := 16#7890ABCD;
END_VAR
TEST('Test_ANY_DWORD_Equals');

AssertEquals(Expected := a,
             Actual := b,
             Message := 'Values differ');

TEST_FINISHED();
END_METHOD

METHOD PRIVATE Test_ANY_INT_Differ
VAR
    a : INT := -32000;
    b : INT := 15423;
END_VAR
TEST('Test_ANY_INT_Differ');

AssertEquals(Expected := a,
             Actual := b,
             Message := 'Values differ');

TEST_FINISHED();
END_METHOD

METHOD PRIVATE Test_ANY_INT_Equals
VAR
    a : INT := -12345;
    b : INT := -12345;
END_VAR
TEST('Test_ANY_INT_Equals');

AssertEquals(Expected := a,
             Actual := b,
             Message := 'Values differ');

TEST_FINISHED();
END_METHOD

METHOD PRIVATE Test_ANY_LINT_Differ
VAR
    a : LINT := -451416345;
    b : LINT := 589532453;
END_VAR
TEST('Test_ANY_LINT_Differ');

AssertEquals(Expected := a,
             Actual := b,
             Message := 'Values differ');

TEST_FINISHED();
END_METHOD

METHOD PRIVATE Test_ANY_LINT_Equals
VAR
    a : LINT := -123456789;
    b : LINT := -123456789;
END_VAR
TEST('Test_ANY_LINT_Equals');

AssertEquals(Expected := a,
             Actual := b,
             Message := 'Values differ');

TEST_FINISHED();
END_METHOD

METHOD PRIVATE Test_ANY_LREAL_Differ
VAR
    a : LREAL := 1234567.89;
    b : LREAL := 1234567.76;
    c : LREAL := 0.0;
END_VAR
TEST('Test_ANY_LREAL_Differ');

AssertEquals(Expected := a,
             Actual := b,
             Message := 'Values a and b differ');

MEMSET (ADR(c), 255, SIZEOF(c));

AssertEquals(Expected := a,
             Actual := c,
             Message := 'Values a and c differ');

TEST_FINISHED();
END_METHOD

METHOD PRIVATE Test_ANY_LREAL_Equals
VAR
    a : LREAL := 1234567.89;
    b : LREAL := 1234567.89;
END_VAR
TEST('Test_ANY_LREAL_Equals');

AssertEquals(Expected := a,
             Actual := b,
             Message := 'Values differ');

TEST_FINISHED();
END_METHOD

METHOD PRIVATE Test_ANY_LTIME_Differ
VAR
    a : LTIME := LTIME#213503D23H34M33S709MS551US615NS;
    b : LTIME := LTIME#1000D15H23M12S34MS2US44NS;
END_VAR
TEST('Test_ANY_LTIME_Differ');

AssertEquals(Expected := a,
             Actual := b,
             Message := 'Values differ');

TEST_FINISHED();
END_METHOD

METHOD PRIVATE Test_ANY_LTIME_Equals
VAR
    a : LTIME := LTIME#213503D23H34M33S709MS551US615NS;
    b : LTIME := LTIME#213503D23H34M33S709MS551US615NS;
END_VAR
TEST('Test_ANY_LTIME_Equals');

AssertEquals(Expected := a,
             Actual := b,
             Message := 'Values differ');

TEST_FINISHED();
END_METHOD

METHOD PRIVATE Test_ANY_LWORD_Differ
VAR
    a : LWORD := 16#0123656789ABCBEC;
    b : LWORD := 16#0123256789ABCAEE;
END_VAR
TEST('Test_ANY_LWORD_Differ');

AssertEquals(Expected := a,
             Actual := b,
             Message := 'Values differ');

TEST_FINISHED();
END_METHOD

METHOD PRIVATE Test_ANY_LWORD_Equals
VAR
    a : LWORD := 16#0123456789ABCDEF;
    b : LWORD := 16#0123456789ABCDEF;
END_VAR
TEST('Test_ANY_LWORD_Equals');

AssertEquals(Expected := a,
             Actual := b,
             Message := 'Values differ');

TEST_FINISHED();
END_METHOD

METHOD PRIVATE Test_ANY_REAL_Differ
VAR
    a : REAL := 1234.5;
    b : REAL := 1234.4;
    c : LREAL := 0.0;
END_VAR
TEST('Test_ANY_REAL_Differ');

AssertEquals(Expected := a,
             Actual := b,
             Message := 'Values a and b differ');

MEMSET (ADR(c), 255, SIZEOF(c));

AssertEquals(Expected := a,
             Actual := c,
             Message := 'Values a and c differ');

TEST_FINISHED();
END_METHOD

METHOD PRIVATE Test_ANY_REAL_Equals
VAR
    a : REAL := 1234.5;
    b : REAL := 1234.5;
END_VAR
TEST('Test_ANY_REAL_Equals');

AssertEquals(Expected := a,
             Actual := b,
             Message := 'Values differ');

TEST_FINISHED();
END_METHOD

METHOD PRIVATE Test_ANY_SINT_Differ
VAR
    a : SINT := 127;
    b : SINT := -30;
END_VAR
TEST('Test_ANY_SINT_Differ');

AssertEquals(Expected := a,
             Actual := b,
             Message := 'Values differ');

TEST_FINISHED();
END_METHOD

METHOD PRIVATE Test_ANY_SINT_Equals
VAR
    a : SINT := -128;
    b : SINT := -128;
END_VAR
TEST('Test_ANY_SINT_Equals');

AssertEquals(Expected := a,
             Actual := b,
             Message := 'Values differ');

TEST_FINISHED();
END_METHOD

METHOD PRIVATE Test_ANY_STRING_Differ
VAR
    a : STRING := 'This is a string';
    b : STRING := 'This is another string';
END_VAR
TEST('Test_ANY_STRING_Differ');

AssertEquals(Expected := a,
             Actual := b,
             Message := 'Values differ');

